// TwinCAT 3 PLC project StandardLibGema
// Title: StandardLibGema
// Company: Gema
// Author: RG
// ProjectVersion: 0.0.83
// ProgramVersion: 3.1.4024.0
// libraries:
//   RFID universal data interface TwinCAT, * (Turck)
//   Tc2_EtherCAT, * (Beckhoff Automation GmbH)
//   Tc2_Standard, * (Beckhoff Automation GmbH)
//   Tc2_System, * (Beckhoff Automation GmbH)
//   Tc2_TcpIp, * (Beckhoff Automation GmbH)
//   Tc2_Utilities, * (Beckhoff Automation GmbH)
//   Tc3_Module, * (Beckhoff Automation GmbH)
//   TcoCore, 0.11.0.71 (Vortex.Library)
//   TcoData, 0.11.0.71 (Vortex.Library)
//   TcoDrivesBeckhoff, 0.11.0.71 (Vortex.Library)
//   TcoElements, 0.11.0.71 (Vortex.Library)
//   TcoIo, 0.11.0.71 (Vortex.Library)
//   TcoPneumatics, 0.11.0.71 (Vortex.Library)
//   TcoUtilities, 0.11.0.71 (Vortex.Library)
//   TcUnit, * (www.tcunit.org)
//   BASIC,3.31,OSCAT
// project tree:
//   IAI/Data types/ AxisLimits.TcDUT, IAIAxisStatus.TcDUT, IOAxis.TcDUT (not stored)
//   IAI/Data types/Enum/ eSetPositionMode.TcDUT (not stored), E_AccelMode.TcDUT, E_RMod.TcDUT, E_StopMode.TcDUT
//   IAI/Data types/Interfaces/ iSuperActuator.TcIO (not stored)
//   IAI/Data types/In/Gateway/ GatewayStatus.TcDUT (not stored), StatusSignal0.TcDUT (not stored), StatusSignal1.TcDUT (not stored)
//   IAI/Data types/In/ PlcIn.TcDUT (not stored), StatusIn.TcDUT (not stored)
//   IAI/Data types/Out/ ControlOut.TcDUT (not stored), PlcOut.TcDUT (not stored)
//   IAI/Data types/Out/Gateway/ ControlSignal0.TcDUT (not stored), ControlSignal1.TcDUT (not stored), GatewayControl.TcDUT
//   IAI/Global Variables/ AxisStats.TcGVL (not stored), AxisStatsGlobal.TcGVL (not stored)
//   IAI/IAI_Drive/TcoAxis/ AxisIAI.TcPOU (not stored), IAxisIAI.TcIO (not stored), Power.TcPOU (not stored)
//   IAI/IAI_Drive/TcoAxis/AxisTasks/ ResetTask.TcPOU (not stored), SetPositionTask.TcPOU (not stored)
//   IAI/IAI_Drive/TcoAxis/MotionTasks/ HaltTask.TcPOU (not stored), HomeTask.TcPOU (not stored), MoveAbsoluteTask.TcPOU (not stored), MoveRelativeTask.TcPOU (not stored), StopTask.TcPOU (not stored)
//   / PlcTask.TcTTO
//   POUs/ATS400_ETL/DUT/ InputDataAts400.TcDUT, State.TcDUT
//   POUs/ATS400_ETL/FunctionBlocks/ InputAts400.TcPOU, OutputAts400.TcPOU, SelectProgramTask.TcPOU
//   POUs/ATS400_ETL/Interfaces/ IInputAts400.TcIO, IOutputAts400.TcIO
//   POUs/ATS400_ETL/Mocks/ InputAts400MockStatusReady.TcPOU
//   POUs/Communication Extern/DUTs/ E_ConnectionStepsTcp.TcDUT, OutCommunicationRobOmron.TcDUT, InCommunicationRobOmron.TcDUT, stTelegrammOmronTcp.TcDUT, uTelegrammOmronTcp.TcDUT
//   POUs/Communication Extern/FunctionBlocks/ CommunicationRoboterOmron.TcPOU, TcpIpCommSeq.TcPOU
//   POUs/Communication Extern/Interfaces/ ICommunicationRoboterOmron.TcIO, ICommSeq.TcIO
//   POUs/Counter Allgemein/ Counter.TcPOU, ICounter.TcIO, StatusCounter.TcDUT
//   POUs/Cylinders/Base/ TcoCylinderBase.TcPOU, TcoDoubleCylinderBase.TcPOU
//   POUs/Cylinders/ExampleCylinder/ ExampleCylinder.TcPOU, ExampleCylinderConfig.TcDUT, ExampleCylinderMoveTask.TcPOU, ExampleCylinderStatus.TcDUT
//   POUs/Cylinders/ ITcoCylinder.TcIO, TcoCylinder.TcPOU, TcoCylinderConfig.TcDUT, TcoCylinderMoveTask.TcPOU, TcoCylinderStatus.TcDUT, TcoDoubleCylinder.TcPOU
//   POUs/Cylinders/Zylinder/ CylCustom.TcPOU, CylCustomMoveTask.TcPOU
//   POUs/DualPositionActuator/DUTs/ E_DualPositionActuatorState.TcDUT
//   POUs/DualPositionActuator/ITFs/ I_DualPositionActuator.TcIO
//   POUs/DualPositionActuator/POUs/ FB_DualPositionActuator.TcPOU
//   POUs/Engel Ethercat Bridge Communication/DUTs/ eHeartBeatState.TcDUT, EngelInputData.TcDUT
//   POUs/Engel Ethercat Bridge Communication/FunctionBlocks/ EngelInput.TcPOU, EngelOutput.TcPOU, HeartBeat.TcPOU, IHeartBeat.TcIO, IInput.TcIO, IOutput.TcIO
//   POUs/Sequences/Test/ E_SequenceTest.TcDUT, SequenceTryout.TcPOU, stSequenceTest.TcDUT
//   POUs/SignalLights MachineStatus/DUTs/ ColorsSignalLightsStatus.TcDUT, eMachineModes.TcDUT, ColorsSignalLightMachineModes.TcDUT, eMachineStatus.TcDUT
//   POUs/SignalLights MachineStatus/ITFs/ ISignalLightsController.TcIO
//   POUs/SignalLights MachineStatus/POUs/ SignalLightsController.TcPOU
//   POUs/Turck Rfid Reader/Mock/ RfidMockNoRfidInRange.TcPOU, RfidMockWorking.TcPOU
//   POUs/Turck Rfid Reader/Rfid/ RfidHead.TcPOU, RfidInOut.TcDUT
//   POUs/Turck Rfid Reader/Rfid/Tasks/ LockTask.TcPOU, ReadDataTask.TcPOU, ReadUidTask.TcPOU, ResetTaskRfid.TcPOU, WriteDataTask.TcPOU
//   POUs/Turck Rfid Reader/Rfid/Wrapper/ IRfidHeadWrapper.TcIO, Rfid_FB_Compact_Wrapper.TcPOU
//   POUs/Utilities/ Blinker.TcPOU
//   Project Information/ F_GetCompany.TcPOU, F_GetTitle.TcPOU, F_GetVersion.TcPOU
//   Test/0 Context/ PRG_TEST.TcPOU, TcUnitContext.TcPOU, TestStation.TcPOU
//   Test/Ats400_Etl_Tests/ InputAts400_Test.TcPOU, OutputAts400_Test.TcPOU
//   Test/BlinkerTest/ Blinker_Test.TcPOU
//   Test/CommunicationExtern Tests/ CommunicationRoboterOmron_Test.TcPOU
//   Test/CounterAllgemeinTests/ Counter_Test.TcPOU
//   Test/DualPositionActuator/ FB_DualPositionActuator_Test.TcPOU
//   Test/Engel Ethercat Bridge Comm Tests/ EngelInput_Test.TcPOU, EngelOutput_Test.TcPOU, HeartBeat_Test.TcPOU
//   Test/Sequences/Test/ SequenceTryout_Test.TcPOU
//   Test/SignalLights MachineStatus Tests/ SignalLightsController_Test.TcPOU
//   Test/Turck Rfid Reader Test/ RfidHead_Test.TcPOU
//   Test/Zylinder Tests/ CylCustom_Test.TcPOU
//   Version/ Global_Version.TcGVL
// real-time tasks:
//   TASK PlcTask: cycle T#1ms, priority 20, ADS port 350

CONFIGURATION StandardLibGema
    RESOURCE PLC ON TwinCAT3
        TASK PlcTask(INTERVAL := T#1ms, PRIORITY := 20);
        PROGRAM PRG_TEST WITH PlcTask : PRG_TEST;
    END_RESOURCE
END_CONFIGURATION

// ---- IAI/Data types/AxisLimits.TcDUT
TYPE
    AxisLimits :
    STRUCT
        MaxAcceleration : UINT;
        MINPosition     : DINT;
        MaxPosition     : DINT;
        MaxVelocity     : UINT;
    END_STRUCT
END_TYPE

// ---- IAI/Data types/Enum/E_AccelMode.TcDUT
//(*Operating mode selector: The AUTO mode is selected when this
//	 signal is OFF, and the MANU mode is selected when the signal is ON*)
TYPE
    E_AccelMode :
    (
        AMode_Trapetz    := 0, (*default*)
        AMode_S_Shape    := 1,
        AMode_FirstOrder := 2
    );
END_TYPE

// ---- IAI/Data types/Enum/E_RMod.TcDUT
//(*Operating mode selector: The AUTO mode is selected when this
//	 signal is OFF, and the MANU mode is selected when the signal is ON*)
TYPE
    E_RMod :
    (
        RMode_Auto := 0,
        RMode_Manu := 1
    );
END_TYPE

// ---- IAI/Data types/Enum/E_StopMode.TcDUT
//(*Operating mode selector: The AUTO mode is selected when this
//	 signal is OFF, and the MANU mode is selected when the signal is ON*)
TYPE
    E_StopMode :
    (
        SMode_OFF      := 0,
        SMode_Param_36 := 1,
        SMode_Param_37 := 2,
        SMode_Param_38 := 3
    );
END_TYPE

// ---- IAI/Data types/IAIAxisStatus.TcDUT
{attribute wpf [Container(Layout.Wrap)]}
TYPE
    IAIAxisStatus :
    STRUCT
        {attribute wpf [Container(Layout.Stack)]}
        {attribute addProperty Name "<#Actual position in mm#>"}
        ActPos : LREAL; (* Actual position (absolut value from NC) *)
        //        {attribute addProperty Name "<#Actual modulo position#>"}
        //        ModuloActPos : LREAL; (* Actual modulo position *)
        //        {attribute addProperty Name "<#Actual modulo turns#>"}
        //        ModuloActTurns : DINT; (* Actual modulo turns *)
        {attribute addProperty Name "<#Actual velocity#>"}
        ActVelo : LREAL; (* Actual velocity *)
        {attribute addProperty Name "<#Actual acceleration#>"}
        ActAcc : LREAL;
        {attribute addProperty Name "<#Actual torque#>"}
        ActTorque : LREAL;
        //        {attribute addProperty Name "<#Command number#>"}
        //        CmdNo : WORD; (* Continuous actual command number *)
        //        {attribute addProperty Name "<#Command state#>"}
        //        CmdState : WORD; (* Command state *)
        //        {attribute addProperty Name "<#Motion state#>"}
        //        MotionState : eAxisStates; (* motion state in the PLCopen state diagram *)
        {attribute addProperty Name "<#Error#>"}
        Error : BOOL; (* axis error state *)
        {attribute addProperty Name "<#Error id#>"}
        ErrorId : UDINT; (* axis error code *)

        (* PLCopen motion control statemachine states: *)
        //        ErrorStop : BOOL;
        //        Disabled : BOOL;
        //        Stopping : BOOL;
        StandStill       : BOOL;
        DiscreteMotion   : BOOL;
        ContinuousMotion : BOOL;
        AbsoluteMotion   : BOOL;
        RelativeMotion   : bool;
        //        SynchronizedMotion : BOOL;
        Homing : BOOL;

        (* additional status - (PLCopen definition)*)
        //        ConstantVelocity : BOOL;
        //        Accelerating : BOOL;
        //        Decelerating : BOOL;

        (* Axis.NcToPlc.StateDWord *)
        Operational : BOOL;
        //        ControlLoopClosed : BOOL; (* operational and position control active *)
        //        HasJob : BOOL;
        HasBeenStopped : BOOL;
        //        NewTargetPosition : BOOL; (* new target position commanded during move *)
        {attribute wpf [Container(Layout.Stack)]}
        InPositionArea    : BOOL;
        InTargetPosition1 : BOOL;
        InTargetPosition2 : BOOL;

        Homed : BOOL;
        //        HomingBusy : BOOL;
        //        MotionCommandsLocked : BOOL; (* stop 'n hold *)
        //        SoftLimitMinExceeded : BOOL; (* reverse soft travel limit exceeded *)
        //        SoftLimitMaxExceeded : BOOL; (* forward soft travel limit exceeded *)

        Moving            : BOOL;
        PositiveDirection : BOOL;
        NegativeDirection : BOOL;
        NotMoving         : BOOL;
        //        Compensating : BOOL; (* superposition - overlayed motion *)

        //        ExtSetPointGenEnabled : BOOL;
        //        ExternalLatchValid : BOOL;
        //        CamDataQueued : BOOL;
        //        CamTableQueued : BOOL;
        //        CamScalingPending : BOOL;
        //        CmdBuffered : BOOL;
        //        PTPmode : BOOL;
        DriveDeviceError : BOOL;
        IoDataInvalid    : BOOL;

        (* Axis.NcToPlc.CoupleState *)
        Coupled1 : BOOL;
        Coupled2 : BOOL;
        Coupled3 : BOOL;
        Coupled4 : BOOL;

    //        (* axis operation mode feedback from NcToPlc *)
    //        OpMode : TcoAxisOpModes;
    END_STRUCT
END_TYPE

// ---- IAI/Data types/Out/Gateway/GatewayControl.TcDUT
TYPE
    GatewayControl :
    STRUCT
        GatewayControl0 : ControlSignal0;
        GatewayControl1 : ControlSignal1;
        RequestCmd      : WORD;
        Data0           : WORD;
        Data1           : WORD;
        Data2           : WORD;
        Data3           : WORD;
        UsedSpace       : WORD;
    END_STRUCT
END_TYPE

// ---- POUs/ATS400_ETL/DUT/InputDataAts400.TcDUT
TYPE
    InputDataAts400 :
    STRUCT
        Pass         : BOOL;
        Fail         : BOOL;
        InOp         : BOOL; // Digitale AUsgabe als Feedback einer aktiven sicherheitstechnischen Pruefung des Systems. Wechselt zwischen dne Pruefungen zwischen 1 auf 0
        ResultImpuls :
            BOOL; // Einstellbare digitale Ausgavbe eines Impuls. Z.B. Gesamtergebnis schlecht, Gesamtergebnis gut etc.
        DummyOut :
            BOOL; //Anofrderung Dummypruefung durch SPS, wartet auf weiteres Feeedback bis Dummy-Pruefobjekt bereit ist
        Ready :
            BOOL;             // wartet auf Start
        SafetyCircuit : BOOL; // 1 = closed, 0 = Open, oder externes Relais, Anzugs- oder Abfallzeit <= 200ms !!
        ContactExits  : BOOL; // Kontaktueberwachung, 1 = Kontakt vorhanden, oder externes Relais
    END_STRUCT
END_TYPE

// ---- POUs/ATS400_ETL/DUT/State.TcDUT
{attribute 'qualified_only'}
{attribute 'strict'}
TYPE
    State :
    (
        Ready := 0,
        Busy,
        Done,
        Fail
    );
END_TYPE

// ---- POUs/Communication Extern/DUTs/E_ConnectionStepsTcp.TcDUT
TYPE
    E_ConnectionStepsTcp :
    (
        eCONNECTION_STATE_IDLE,
        eCONNECTION_STATE_CONNECT_START,
        eCONNECTION_STATE_CONNECT_WAIT,
        eCONNECTION_STATE_DATAEXCHANGE,
        eCONNECTION_STATE_CLOSE_START,
        eCONNECTION_STATE_CLOSE_WAIT,
        eCONNECTION_STATE_ERROR
    );
END_TYPE

// ---- POUs/Communication Extern/DUTs/OutCommunicationRobOmron.TcDUT
TYPE
    OutCommunicationRobOmron :
    STRUCT
        {attribute addProperty Name "<#AutoMode Aktiv#>"}
        StartAutomatic  : BOOL;
        StopAutomatic   : BOOL;
        Reset           : BOOL;
        RequestHome     : BOOL;
        HighPowerOn     : BOOL;
        HighPowerOff    : BOOL;
        ContactPrepared : BOOL;
    END_STRUCT
END_TYPE

// ---- POUs/Communication Extern/DUTs/InCommunicationRobOmron.TcDUT
TYPE
    InCommunicationRobOmron :
    STRUCT
        {attribute addProperty Name "<#Home Pos erreicht#>"}
        homePosReached : BOOL;
        {attribute addProperty Name "<#Status Running#>"}
        statusRunning : BOOL;
        {attribute addProperty Name "<#Fehler#>"}
        Fault : BOOL;
        {attribute addProperty Name "<#Fehler ID#>"}
        FaultID : INT;
        {attribute addProperty Name "<#HighPower aktiv#>"}
        PowerOn : BOOL;
        {attribute addProperty Name "<#EStop aktiv#>"}
        Estop : BOOL;
    END_STRUCT
END_TYPE

// ---- POUs/Communication Extern/DUTs/stTelegrammOmronTcp.TcDUT
{attribute 'pack_mode' := '1'}
TYPE
    stTelegrammOmronTcp :
    STRUCT
        myStats  : ARRAY[1..4] OF BYTE;
        myInt    : ARRAY[1..10] OF INT;
        myBool   : ARRAY[1..20] OF INT;
        fillbyte : ARRAY[1..2] OF BYTE;
    END_STRUCT
END_TYPE

// ---- POUs/Communication Extern/DUTs/uTelegrammOmronTcp.TcDUT
TYPE
    uTelegrammOmronTcp :
    UNION
        //~
        stTel : stTelegrammOmronTcp;
        aTel  : ARRAY[1..SIZEOF(stTelegrammOmronTcp)] OF BYTE;
        sTel  : STRING(SIZEOF(stTelegrammOmronTcp));
    //~
    END_UNION
END_TYPE

// ---- POUs/Counter Allgemein/StatusCounter.TcDUT
{attribute 'qualified_only'}
{attribute 'strict'}
TYPE StatusCounter :
(
    Error := 0,
    Run,
    Unknown
);
END_TYPE

// ---- POUs/Cylinders/ExampleCylinder/ExampleCylinderConfig.TcDUT
TYPE
    ExampleCylinderConfig :
    STRUCT
        TimeToReachHomePosition : TIME := T#10S;
        TimeToReachWorkPosition : TIME := T#10S;
    END_STRUCT
END_TYPE

// ---- POUs/Cylinders/ExampleCylinder/ExampleCylinderStatus.TcDUT
TYPE
    ExampleCylinderStatus :
    STRUCT
        ActionDescription : STRING(100);
    END_STRUCT
END_TYPE

// ---- POUs/Cylinders/TcoCylinderConfig.TcDUT
TYPE
    TcoCylinderConfig :
    STRUCT
        TimeToReachHomePosition : TIME := T#10S;
        TimeToReachWorkPosition : TIME := T#10S;
        TimeToRefill            : TIME := T#1000MS;
    END_STRUCT
END_TYPE

// ---- POUs/Cylinders/TcoCylinderStatus.TcDUT
TYPE
    TcoCylinderStatus :
    STRUCT
        ActionDescription : STRING(100);
    END_STRUCT
END_TYPE

// ---- POUs/DualPositionActuator/DUTs/E_DualPositionActuatorState.TcDUT
{attribute 'qualified_only'}
{attribute 'strict'}
{attribute 'to_string'}
TYPE
    E_DualPositionActuatorState :
    (
        Unknown := 0,
        Active,
        Disabled,
        TimeoutActivating,
        TimeoutDisabling,
        Activating,
        Disabling
    ) INT;
END_TYPE

// ---- POUs/Engel Ethercat Bridge Communication/DUTs/eHeartBeatState.TcDUT
{attribute 'qualified_only'}
{attribute 'strict'}
{attribute 'to_string'}
TYPE
    eHeartBeatState :
    (
        Unknown := 0,
        Valid,
        Timeout
    ) INT;
END_TYPE

// ---- POUs/Engel Ethercat Bridge Communication/DUTs/EngelInputData.TcDUT
TYPE
    EngelInputData :
    STRUCT
        HeartBeat            : UINT;
        ManualActive         : BOOL;
        AutoActive           : BOOL;
        AutoStart            : BOOL;
        HomeRequest          : BOOL;
        HomeDone             : BOOL;
        SafetyClosed         : BOOL;
        SafetyOpeningAllowed : BOOL;

    END_STRUCT
END_TYPE

// ---- POUs/Sequences/Test/E_SequenceTest.TcDUT
{attribute 'qualified_only'}
{attribute 'strict'}
{attribute 'to_string'}
TYPE
    E_SequenceTest :
    (
        WaitForStart,
        OpenValveAandB,
        ConfirmValvesAandBOpend,
        CloseValveA,
        ConfirmClosedValveA,
        Error,
        Done
    ) INT;
END_TYPE

// ---- POUs/Sequences/Test/stSequenceTest.TcDUT
TYPE
    stSequenceTest :
    STRUCT
        WaitForStart   : INT := 10;
        OpenValveAandB : INT := 20;
    END_STRUCT
END_TYPE

// ---- POUs/SignalLights MachineStatus/DUTs/ColorsSignalLightsStatus.TcDUT
TYPE
    ColorsSignalLightsStatus :
    STRUCT
        Blue     : BOOL;
        White    : BOOL;
        Violet   : BOOL;
        Turquise : BOOL;
    END_STRUCT
END_TYPE

// ---- POUs/SignalLights MachineStatus/DUTs/eMachineModes.TcDUT
{attribute 'qualified_only'}
{attribute 'strict'}
{attribute 'to_string'}
TYPE
    eMachineModes :
    (
        Idle    := 0,
        Automat := 1000,
        Step    := 2000,
        Home    := 3000,
        Manual  := 4000,
        Fault   := 9000
    ) INT;
END_TYPE

// ---- POUs/SignalLights MachineStatus/DUTs/ColorsSignalLightMachineModes.TcDUT
TYPE
    ColorsSignalLightMachineModes :
    STRUCT
        Green       : BOOL;
        Yellow      : BOOL;
        Red         : BOOL;
    END_STRUCT
END_TYPE

// ---- POUs/SignalLights MachineStatus/DUTs/eMachineStatus.TcDUT
{attribute 'qualified_only'}
{attribute 'strict'}
{attribute 'to_string'}
TYPE
    eMachineStatus :
    (

        Blue     := 100,
        White    := 200,
        Violet   := 300,
        Turquise := 400,
        All      := 990
    ) INT;
END_TYPE

// ---- POUs/Turck Rfid Reader/Rfid/RfidInOut.TcDUT
TYPE
    RfidInOut :
    STRUCT

        myReadData             : ARRAY[0..127] OF BYTE;
        myWriteData            : ARRAY[0..127] OF BYTE;
        xExecute               : BOOL;
        xAbort                 : BOOL;
        udiTimeOut             : UDINT;
        eCommand               : RFID_FB_U.COMMAND;
        udiStartAdress         : UDINT;
        uiDataLenght           : UINT;
        xDone                  : BOOL;
        xBusy                  : BOOL;
        xError                 : BOOL;
        xAborted               : BOOL;
        eErrorID               : RFID_FB_U.ERROR;
        xTP                    : BOOL;
        xRWHeadNotCOnnected    : BOOL;
        uiDataRxLength         : UINT;
        stCompactModeInputMap  : RFID_FB_U.CompactInput_t;
        stCompactModeOutputMap : RFID_FB_U.CompactOutput_t;
    END_STRUCT
END_TYPE

// ---- Version/Global_Version.TcGVL
{attribute 'TcGenerated'}
{attribute 'no-analysis'}
{attribute 'linkalways'}
// This function has been automatically generated from the project information.
VAR_GLOBAL CONSTANT
    {attribute 'const_non_replaced'}
    stLibVersion_StandardLibGema : ST_LibVersion :=
    (
        iMajor      := 0
        , iMinor    := 0
        , iBuild    := 83
        , iRevision := 0
        , nFlags    := 0
        , sVersion  := '0.0.83'
    );
END_VAR

// ---- POUs/ATS400_ETL/Interfaces/IInputAts400.TcIO
INTERFACE IInputAts400 EXTENDS __SYSTEM.IQueryInterface

METHOD GetInputData : InputDataAts400
VAR_INPUT
END_VAR
END_METHOD

END_INTERFACE

// ---- POUs/ATS400_ETL/Interfaces/IOutputAts400.TcIO
INTERFACE IOutputAts400 EXTENDS __SYSTEM.IQueryInterface

METHOD AbortTest
VAR_INPUT
    enable : BOOL;
END_VAR
END_METHOD

METHOD SelectProgramm : TcoCore.ITcoTaskStatus
VAR_INPUT
    programm : UINT;
END_VAR
END_METHOD

METHOD SetDummyReady
VAR_INPUT
    enable : BOOL;
END_VAR
END_METHOD

METHOD SetManualFail
VAR_INPUT
    enable : BOOL;
END_VAR
END_METHOD

METHOD SetManualPass
VAR_INPUT
    enable : BOOL;
END_VAR
END_METHOD

METHOD Start
VAR_INPUT
    enable : BOOL;
END_VAR
END_METHOD

END_INTERFACE

// ---- POUs/Communication Extern/Interfaces/ICommunicationRoboterOmron.TcIO
INTERFACE ICommunicationRoboterOmron EXTENDS __SYSTEM.IQueryInterface

METHOD ContactPrepared
VAR_INPUT
    enable : BOOL;
END_VAR
END_METHOD

PROPERTY EState : E_SocketConnectionState
GET
END_GET
END_PROPERTY

METHOD HighPowerOn
VAR_INPUT
    enable : BOOL;
END_VAR
END_METHOD

PROPERTY MsgFmtStr : T_MaxString
GET
END_GET
END_PROPERTY

METHOD RequestHome
VAR_INPUT
    enable : BOOL;
END_VAR
END_METHOD

METHOD Reset
VAR_INPUT
    enable : BOOL;
END_VAR
END_METHOD

METHOD Run
END_METHOD

METHOD StartAutomatic
VAR_INPUT
    enable : BOOL;
END_VAR
END_METHOD

METHOD StopAutomatic
VAR_INPUT
    enable : BOOL;
END_VAR
END_METHOD

END_INTERFACE

// ---- POUs/Communication Extern/Interfaces/ICommSeq.TcIO
INTERFACE ICommSeq

PROPERTY EState : E_SocketConnectionState
GET
END_GET
END_PROPERTY

PROPERTY MsgFmtStr : T_MaxString
GET
END_GET
END_PROPERTY

METHOD Run
VAR_INPUT
    msgSend : REFERENCE TO uTelegrammOmronTcp;
    msgRcv  : REFERENCE TO uTelegrammOmronTcp;
END_VAR
END_METHOD

END_INTERFACE

// ---- POUs/Counter Allgemein/ICounter.TcIO
INTERFACE ICounter

METHOD CountDown
END_METHOD

PROPERTY CountLimitReached : BOOL
GET
END_GET
END_PROPERTY

METHOD CountUp
VAR_INPUT
END_VAR
END_METHOD

PROPERTY CountValue : UDINT
GET
END_GET
END_PROPERTY

PROPERTY CountZeroReached : BOOL
GET
END_GET
END_PROPERTY

METHOD ResetCount
VAR_INPUT
END_VAR
END_METHOD

END_INTERFACE

// ---- POUs/Cylinders/ITcoCylinder.TcIO
INTERFACE ITcoCylinder EXTENDS __System.IQueryInterface

PROPERTY AtHome : bool
GET
END_GET
END_PROPERTY

PROPERTY AtWork : bool
GET
END_GET
END_PROPERTY

METHOD MoveToHome : TcoCore.ITcoTaskStatus
END_METHOD

METHOD MoveToWork : TcoCore.ITcoTaskStatus
END_METHOD

(*~
	<docu>
		<summary>
			Stops cyclinder movement.
		 	<remarks>
				<note type="important">
					This method switched off the signals for the movement of the piston in both direction.
					However depending on the pnemumatics configuration the movement may contintue if designed in that way.
					THIS IS NOT A SAFETY FUCTION!
				</note>
			</remarks>
		</summary>
	</docu>
~*)
METHOD Stop : TcoCore.ITcoTaskStatus
END_METHOD

END_INTERFACE

// ---- POUs/DualPositionActuator/ITFs/I_DualPositionActuator.TcIO
INTERFACE I_DualPositionActuator

METHOD PUBLIC Activate
END_METHOD

METHOD PUBLIC Disable
END_METHOD

METHOD GetDisableTimeoutTime : TIME
END_METHOD

METHOD GetEnableTimeoutTime : TIME
END_METHOD

METHOD GetState : E_DualPositionActuatorState
END_METHOD

METHOD SetDisableTimeoutTime
VAR_INPUT
    tDisableTimeoutTime : TIME;
END_VAR
END_METHOD

METHOD SetEnableTimeoutTime
VAR_INPUT
    tEnableTimeoutTime : TIME;
END_VAR
END_METHOD

END_INTERFACE

// ---- POUs/Engel Ethercat Bridge Communication/FunctionBlocks/IHeartBeat.TcIO
INTERFACE IHeartBeat EXTENDS __SYSTEM.IQueryInterface

PROPERTY GetErrorMessage : T_MaxString;
GET
END_GET
END_PROPERTY

//actual Heartbeat of PLC
PROPERTY GetHeartBeat : UINT
GET
END_GET
END_PROPERTY

PROPERTY GetHeartbeatTimeoutTime : TIME
GET
END_GET
END_PROPERTY

PROPERTY GetState : eHeartBeatState
GET
END_GET
END_PROPERTY

METHOD IncreaseHeartBeat : UINT
VAR_INPUT
    externalHeartBeat : UINT;
END_VAR
END_METHOD

END_INTERFACE

// ---- POUs/Engel Ethercat Bridge Communication/FunctionBlocks/IInput.TcIO
INTERFACE IInput

METHOD GetInputData : EngelInputData
END_METHOD

END_INTERFACE

// ---- POUs/Engel Ethercat Bridge Communication/FunctionBlocks/IOutput.TcIO
INTERFACE IOutput EXTENDS __SYSTEM.IQueryInterface

END_INTERFACE

// ---- POUs/SignalLights MachineStatus/ITFs/ISignalLightsController.TcIO
INTERFACE ISignalLightsController

PROPERTY GetColorsSignalLightMachineModes : ColorsSignalLightMachineModes
GET
END_GET
END_PROPERTY

PROPERTY GetColorsSignalLightMachineStatus : ColorsSignalLightsStatus
GET
END_GET
END_PROPERTY

METHOD SetBlinkTime
VAR_INPUT
    blinkOnTime  : TIME;
    blinkOffTime : TIME;
END_VAR
END_METHOD

METHOD SetMachineMode : ColorsSignalLightMachineModes
VAR_INPUT
    currentMachineMode : eMachineModes ;
END_VAR
END_METHOD

METHOD SetMachineStatusOff : ColorsSignalLightsStatus
VAR_INPUT
    currentMachineStatus : eMachineStatus ;
END_VAR
END_METHOD

METHOD SetMachineStatusOn : ColorsSignalLightsStatus
VAR_INPUT
    currentMachineStatus : eMachineStatus ;
END_VAR
END_METHOD

END_INTERFACE

// ---- POUs/Turck Rfid Reader/Rfid/Wrapper/IRfidHeadWrapper.TcIO
INTERFACE IRfidHeadWrapper

METHOD Execute
VAR_INPUT
    xExecute       : BOOL;
    xAbort         : BOOL;
    udiTimeOut     : UDINT;
    eCommand       : RFID_FB_U.COMMAND;
    udiStartAdress : UDINT;
    uiDataLenght   : UINT;
    myWriteData    : ARRAY[0..127] OF BYTE;
END_VAR
VAR_OUTPUT
    myReadData          : ARRAY[0..127] OF BYTE;
    xDone               : BOOL;
    xBusy               : BOOL;
    xError              : BOOL;
    xAborted            : BOOL;
    eErrorID            : RFID_FB_U.ERROR;
    xTP                 : BOOL;
    xRWHeadNotCOnnected : BOOL;
    uiDataRxLength      : UINT;
END_VAR
END_METHOD

END_INTERFACE

// ---- Test/0 Context/PRG_TEST.TcPOU
PROGRAM PRG_TEST
VAR
    _testSuite : TcUnitContext;
END_VAR

_testSuite.Run();
_testSuite.RtcSynchronize(true, '', 60);

END_PROGRAM

// ---- Test/0 Context/TcUnitContext.TcPOU
FUNCTION_BLOCK TcUnitContext EXTENDS TcoCore.TcoContext
VAR
    testStation : TestStation(THIS^);

    {attribute addProperty Name "Versionsnummer Plc"}
    version : STRING(23);
    //~
    programVersion : ST_LibVersion;
    //~

END_VAR

(*~
    <docu>
        <summary>
            Main method of the TcoContext. This is the entry point of any control logic that belongs to this context.
            The call of this method is ensured by calling the <c>InstanceName.Run()</c> method, and it must not be called explicitly.
            This method is abstract, and it must be overridden in derived block.
        </summary>
    </docu>
~*)
METHOD PROTECTED Main

testStation();
END_METHOD

END_FUNCTION_BLOCK

// ---- Test/0 Context/TestStation.TcPOU
FUNCTION_BLOCK TestStation EXTENDS TcoCore.TcoObject
VAR
    cylCustomTest : CylCustom_Test;
END_VAR
//===============================Turck Rfid Reader===============================================
VAR
    rfidHead_Test : RfidHead_Test;
END_VAR
//===================================================================================

//====================== Engel Communication Ethercat Bridge =====================================
VAR
    engelInputTest     : EngelInput_Test;
    engelOutputTest    : EngelOutput_Test;
    engelHeartBeatTest : HeartBeat_Test;
END_VAR
//===================================================================================

//===============================Dual Position Actuator Sagatowski===============================================
VAR
    sequenceTryOutTest : SequenceTryout_Test;
END_VAR
//====
//===============================Dual Position Actuator Sagatowski===============================================
VAR
    dualPositionActuator_Test : FB_DualPositionActuator_Test;
END_VAR
//===================================================================================

//===============================Communication with ETL ATS400 ===============================================
VAR
    inputAts400Test  : InputAts400_Test;
    outputAts400Test : OutputAts400_Test;
END_VAR
//===================================================================================
//===============================Communication with ETL ATS400 ===============================================
VAR
    CommunicationRoboterOmron  : CommunicationRoboterOmron_Test;

END_VAR
//===================================================================================
//===============================SignalLights for MachineStatus ===============================================
VAR
    signalLightsControllerTest : SignalLightsController_Test;
END_VAR
//===================================================================================
//===============================Utilities ===============================================
VAR
    blinkerTest : Blinker_Test;
    counterTest : Counter_Test;
END_VAR
//=======

TcUnit.RUN();

END_FUNCTION_BLOCK

// ---- Test/Zylinder Tests/CylCustom_Test.TcPOU
FUNCTION_BLOCK CylCustom_Test EXTENDS TcUnit.FB_TestSuite IMPLEMENTS TcoCore.ITcoContext
VAR
    //Context for TcOpen
    _nfContext : TcoCore.TcoContextNfCompatibility;
END_VAR

VAR
    fbTestTimer : TON := (PT := T#30ms);
    cyl         : TcoCylinder(THIS^);
    sensor      : ARRAY[0..1] OF BOOL;
    actuator    : ARRAY[0..1] OF BOOL;
    nTestState  : INT;
END_VAR

_nfContext.VolatileOpen(); //Required for TCopen
//==============================================

ExecuteMoveToWork_SignalAtWorkShouldBeTrue();

//==============================================
_nfContext.VolatileClose();

PROPERTY Context : TcoCore.ITcoContext
GET
Context := This^._nfContext;
END_GET
END_PROPERTY

PROPERTY EndCycleCount : ULINT
GET
EndCycleCount := THIS^._nfContext._endCycleCount;
END_GET
END_PROPERTY

PROPERTY Environment : TcoCore.ITcoContextEnvironment
GET
Environment := THIS^._nfContext._settings;
END_GET
END_PROPERTY

METHOD PRIVATE ExecuteMoveToWork_SignalAtWorkShouldBeTrue
Test('ExecuteMoveToWork_SignalAtWorkShouldBeTrue');
fbTestTimer(IN := TRUE);
cyl
(
    inoAtHomePos   := sensor[0]
    , inoAtWorkPos := sensor[1]
    , inoToHomePos := actuator[0]
    , inoToWorkPos := actuator[1]
);

CASE nTestState OF
    0:
        sensor[0]  := TRUE;
        nTestState := nTestState + 1;
    1:
        // Retracted
        AssertTrue(cyl.AtHome, 'Should be AtHome');
        nTestState := nTestState + 1;
    2:
        sensor[0] := FALSE;
        cyl.MoveToWork();
        nTestState := nTestState + 1;
    3:
        AssertTrue(actuator[1], 'should turn True');
        nTestState := nTestState + 1;
    4:
        sensor[1]  := TRUE;
        nTestState := nTestState + 1;
    5:
        AssertTrue(cyl.AtWork, 'should reach Work');
END_CASE

IF fbTestTimer.Q THEN
    Assertequals_INT(Expected := 5, Actual := nTestState, Message := 'Didnt reach the last state');
    TEST_FINISHED();
END_IF
END_METHOD

PROPERTY Identity : ULINT
GET
Identity := THIS^._nfContext._Identity;
END_GET
END_PROPERTY

PROPERTY Logger : TcoCore.ITcoLogger
GET
Logger := THIS^._nfContext._logger;
END_GET
END_PROPERTY

PROPERTY RealTimeClock : TcoCore.ITcoRtc
GET
RealTimeClock := THIS^._nfContext._rtc;
END_GET
END_PROPERTY

PROPERTY StartCycleCount : ULINT
GET
StartCycleCount := THIS^._nfContext._startCycleCount;
END_GET
END_PROPERTY

END_FUNCTION_BLOCK

// ---- POUs/Cylinders/TcoCylinder.TcPOU
{attribute addProperty _moveHomeDefaultName "<#MOVE HOME#>"}
{attribute addProperty _moveWorkDefaultName "<#MOVE TO WORK#>"}
{attribute addProperty _stopDefaultName "<#STOP#>"}
FUNCTION_BLOCK TcoCylinder EXTENDS TcoCylinderBase
VAR
    {attribute addProperty Name "|[[1]Attribute_moveHomeDefaultName]|"}
    _moveHomeDefault : TcoCylinderMoveTask(THIS^);
    {attribute addProperty Name "|[[1]Attribute_moveWorkDefaultName]|"}
    _moveWorkDefault : TcoCylinderMoveTask(THIS^);
    {attribute addProperty Name "|[[1]Attribute_stopDefaultName]|"}
    _stopDefault : TcoCore.TcoTask(THIS^);
    increment    : INT;
END_VAR
VAR
    _config      : TcoCylinderConfig;
    _status      : TcoCylinderStatus;
    _refillTimer : TON;
END_VAR

SUPER^
(
    inoAtHomePos   := inoAtHomePos
    , inoAtWorkPos := inoAtWorkPos
    , inoToHomePos := inoToHomePos
    , inoToWorkPos := inoToWorkPos
);

IF (_atHomePos AND _atWorkPos) THEN
    Messenger.Error('<#Home and work position sensors are both active. Check the position of sensors!#>');
END_IF;

// Disables mutualy exclusive actions
_moveWorkDefault.Enabled := TRUE; // NOT _moveHomeDefault.Busy;

_moveHomeDefault
(
    PositionSensor           := _atHomePos AND NOT _atWorkPos
    , MoveToPositionSignal   := _toHomePos
    , InverseSignal          := _toWorkPos
    , TimeToRefill           := _config.TimeToRefill
    , MaxTimeToReachPosition := _config.TimeToReachHomePosition
    , PositionName           := '<#Home#>'
);

IF _moveHomeDefault.Execute() THEN
    _moveWorkDefault.Restore();
END_IF

// Disables mutualy exclusive actions
_moveHomeDefault.Enabled := TRUE; //NOT _moveWorkDefault.Busy;

_moveWorkDefault
(
    PositionSensor           := _atWorkPos AND NOT _atHomePos
    , MoveToPositionSignal   := _toWorkPos
    , InverseSignal          := _toHomePos
    , TimeToRefill           := _config.TimeToRefill
    , MaxTimeToReachPosition := _config.TimeToReachWorkPosition
    , PositionName           := '<#Work#>'
);

IF _moveWorkDefault.Execute() THEN
    _moveHomeDefault.Restore();
END_IF

IF (_stopDefault.Execute()) THEN
    _toHomePos := FALSE;
    _toWorkPos := FALSE;
    _moveHomeDefault.Abort();
    _moveWorkDefault.Abort();
    _stopDefault.Abort();
    _moveHomeDefault.Restore();
    _moveWorkDefault.Restore();
    _stopDefault.Restore();
    _stopDefault.DoneWhen(TRUE);
END_IF

// For further discussion about Status
IF (_moveHomeDefault.Busy) THEN
    _status.ActionDescription := 'Moving to home position';
ELSIF (_moveWorkDefault.Busy) THEN
    _status.ActionDescription := 'Moving to work position';
ELSIF (_stopDefault.Busy) THEN
    _status.ActionDescription := 'Stopping pressure';
ELSE
    _status.ActionDescription := 'Idle';
END_IF

SUPER^
(
    inoAtHomePos   := inoAtHomePos
    , inoAtWorkPos := inoAtWorkPos
    , inoToHomePos := inoToHomePos
    , inoToWorkPos := inoToWorkPos
);

(*~
    <docu>
        <summary>
            Aborts the movement to home position when the condition is 'true'.
        </summary>
        <remarks>
                <note type="warning">
                    The call of this method will be effective only when called AFTER the initialization of the instance of given TcoCylinder.
                </note>
        </remarks>
    </docu>
~*)
METHOD AbortMoveHome : BOOL
VAR_IN_OUT
    (*~
    <docu>
        <summary>
            Condition to abort the movement of the cylinder.
        </summary>
    </docu>
    ~*)
    inoDisableCondition : BOOL;
END_VAR
VAR
    _signalInfo : TcoSignalInfo;
END_VAR
IF (_toHomePos OR _moveHomeDefault.Busy) AND inoDisableCondition THEN
    _signalInfo.GetSignalInfo(SIZEOF(inoDisableCondition), ADR(inoDisableCondition));
    Messenger.Build().Append('<#Movement aborted due to#> : ').Append(_signalInfo.SymbolPath).As().AsError().Pin();
    _toHomePos := FALSE;
    IF (__ISVALIDREF(THIS^.inoToHomePos)) THEN
        THIS^.inoToHomePos := FALSE;
    END_IF;

    _moveHomeDefault.Abort();
END_IF
END_METHOD

(*~
    <docu>
        <summary>
            Aborts the movement to work position when the condition is 'true'.
        </summary>
        <remarks>
                <note type="warning">
                    The call of this method will be effective only when called AFTER the initialization of the instance of given TcoCylinder.
                </note>
        </remarks>
    </docu>
~*)
METHOD AbortMoveWork : BOOL
VAR_IN_OUT
    (*~
        <docu>
            <summary>
                Condition to abort the movement of the cylinder.
            </summary>
        </docu>
    ~*)
    inoDisableCondition : BOOL;
END_VAR
VAR
    _signalInfo : TcoSignalInfo;
END_VAR
IF (_toWorkPos OR _moveWorkDefault.Busy) AND inoDisableCondition THEN
    _signalInfo.GetSignalInfo(SIZEOF(inoDisableCondition), ADR(inoDisableCondition));
    Messenger.Build().Append('<#Movement aborted due to#> : ').Append(_signalInfo.SymbolPath).As().AsError().Pin();
    _toWorkPos := FALSE;
    IF (__ISVALIDREF(THIS^.inoToWorkPos)) THEN
        THIS^.inoToWorkPos := FALSE;
    END_IF;

    _moveWorkDefault.Abort();
END_IF
END_METHOD

(*~
    <docu>
        <summary>
            Gets the configuration of the cylinder.
        </summary>
    </docu>
~*)
PROPERTY Config : REFERENCE TO TcoCylinderConfig
GET
Config REF= _config;
END_GET
END_PROPERTY

(*~
    <docu>
        <summary>
            Gets the `MoveHomeTask` task that controls the moving of the cyclinder in home position.
        </summary>
    </docu>
~*)
PROPERTY MoveHomeTask : TcoCore.ITcoTask
GET
MoveHomeTask := _moveHomeDefault;
END_GET
END_PROPERTY

(*~
    <docu>
        <summary>
            Gets the `MoveWorkTask` task that controls the moving of the cyclinder into work position.
        </summary>
    </docu>
~*)
PROPERTY MoveWorkTask : TcoCore.ITcoTask
GET
MoveWorkTask := _moveWorkDefault;
END_GET
END_PROPERTY

(*~
    <docu>
        <summary>
            Refill cylinder after booth outputs are off .
        </summary>
        <remarks>
                <note type="warning">
                    The call of this method will be effective only when called AFTER the initialization of the instance of given TcoCylinder and methods like AbortMoveHone,SuspendMoveHom...
                </note>
        </remarks>
    </docu>
~*)
METHOD Refill : BOOL
VAR_INPUT
    (*~
    <docu>
        <summary>
            Time of refill cylinder after aborting or suspending
        </summary>
    </docu>
    ~*)
    inRefillTime : TIME;
END_VAR

_refillTimer(In := inoToHomePos XOR inoToWorkPos, Pt := T#49D);

_config.TimeToRefill := inRefillTime;

IF _refillTimer.ET > T#0MS
       AND _refillTimer.ET < _config.TimeToRefill
       AND _config.TimeToRefill <> T#0S THEN
    _toHomePos := TRUE;
    _toWorkPos := TRUE;
END_IF;

SUPER^
(
    inoAtHomePos   := inoAtHomePos
    , inoAtWorkPos := inoAtWorkPos
    , inoToHomePos := inoToHomePos
    , inoToWorkPos := inoToWorkPos
);
END_METHOD

PROPERTY StatusCom : REFERENCE TO TcoCylinderStatus
GET
StatusCom REF= _status;
END_GET
END_PROPERTY

(*~
    <docu>
        <summary>
            Gets the `StopTask` task that controls the stopping of the cyclinder.
        </summary>
    </docu>
~*)
PROPERTY StopTask : TcoCore.ITcoTask
GET
StopTask := _stopDefault;
END_GET
END_PROPERTY

(*~
    <docu>
        <summary>
            Suspend the movement to home position when the condition is 'true'. Task is still busy
        </summary>
        <remarks>
                <note type="warning">
                    The call of this method will be effective only when called AFTER the initialization of the instance of given TcoCylinder.
                </note>
        </remarks>
    </docu>
~*)
METHOD SuspendMoveHome : BOOL
VAR_IN_OUT
    (*~
    <docu>
        <summary>
            Condition to abort the movement of the cylinder.
        </summary>
    </docu>
    ~*)
    inoDisableCondition : BOOL;
END_VAR
VAR
    _signalInfo : TcoSignalInfo;
END_VAR
IF (_toHomePos OR _moveHomeDefault.Busy) AND inoDisableCondition THEN
    _signalInfo.GetSignalInfo(SIZEOF(inoDisableCondition), ADR(inoDisableCondition));
    Messenger.Warning(CONCAT('<#Movement suspended due to#> : ', _signalInfo.SymbolPath));
    _toHomePos := FALSE;
    IF (__ISVALIDREF(THIS^.inoToHomePos)) THEN
        THIS^.inoToHomePos := FALSE;
    END_IF;

END_IF
END_METHOD

METHOD SuspendMoveHomeExpression : BOOL
VAR_INPUT
    inDisableCondition : BOOL;
    inMessage          : STRING;
END_VAR
IF (_toHomePos OR _moveHomeDefault.Busy) AND inDisableCondition THEN
    Messenger.Warning(CONCAT('<#Movement suspended due to#> : ', inMessage));
    _toHomePos := FALSE;
    IF (__ISVALIDREF(THIS^.inoToHomePos)) THEN
        THIS^.inoToHomePos := FALSE;
    END_IF;

END_IF;
END_METHOD

(*~
    <docu>
        <summary>
            Suspend the movement to home position when the condition is NOT 'true'. Task is still busy
        </summary>
        <remarks>
                <note type="warning">
                    The call of this method will be effective only when called AFTER the initialization of the instance of given TcoCylinder.
                </note>
        </remarks>
    </docu>
~*)
METHOD SuspendMoveHomeInverted : BOOL
VAR_IN_OUT
    (*~
    <docu>
        <summary>
            Condition to abort the movement of the cylinder.
        </summary>
    </docu>
    ~*)
    inoDisableCondition : BOOL;
END_VAR
VAR
    _signalInfo : TcoSignalInfo;
END_VAR
IF (_toHomePos OR _moveHomeDefault.Busy) AND not inoDisableCondition THEN
    _signalInfo.GetSignalInfo(SIZEOF(inoDisableCondition), ADR(inoDisableCondition));
    Messenger.Warning(CONCAT('<#Movement suspended due to NOT#> : ', _signalInfo.SymbolPath));
    _toHomePos := FALSE;
    IF (__ISVALIDREF(THIS^.inoToHomePos)) THEN
        THIS^.inoToHomePos := FALSE;
    END_IF;

END_IF
END_METHOD

(*~
    <docu>
        <summary>
            Suspend the movement to work position when the condition is 'true'. Task is still bussy
        </summary>
        <remarks>
                <note type="warning">
                    The call of this method will be effective only when called AFTER the initialization of the instance of given TcoCylinder.
                </note>
        </remarks>
    </docu>
~*)
METHOD SuspendMoveWork : BOOL
VAR_IN_OUT
    (*~
        <docu>
            <summary>
                Condition to abort the movement of the cylinder.
            </summary>
        </docu>
    ~*)
    inoDisableCondition : BOOL;
END_VAR
VAR
    _signalInfo : TcoSignalInfo;
END_VAR
IF (_toWorkPos OR _moveWorkDefault.Busy) AND inoDisableCondition THEN
    _signalInfo.GetSignalInfo(SIZEOF(inoDisableCondition), ADR(inoDisableCondition));
    Messenger.Warning(CONCAT('<#Movement suspended due to#> : ', _signalInfo.SymbolPath));
    _toWorkPos := FALSE;
    IF (__ISVALIDREF(THIS^.inoToWorkPos)) THEN
        THIS^.inoToWorkPos := FALSE;
    END_IF;

END_IF
END_METHOD

METHOD SuspendMoveWorkExpression : BOOL
VAR_INPUT
    inDisableCondition : BOOL;
    inMessage          : STRING;
END_VAR
IF (_toWorkPos OR _moveWorkDefault.Busy) AND inDisableCondition THEN
    Messenger.Warning(CONCAT('<#Movement suspended due to#> : ', inMessage));
    _toWorkPos := FALSE;
    IF (__ISVALIDREF(THIS^.inoToWorkPos)) THEN
        THIS^.inoToWorkPos := FALSE;
    END_IF;

END_IF
END_METHOD

(*~
    <docu>
        <summary>
            Suspend the movement to work position when the condition is NOT 'true'. Task is still busy
        </summary>
        <remarks>
                <note type="warning">
                    The call of this method will be effective only when called AFTER the initialization of the instance of given TcoCylinder.
                </note>
        </remarks>
    </docu>
~*)
METHOD SuspendMoveWorkInverted : BOOL
VAR_IN_OUT
    (*~
        <docu>
            <summary>
                Condition to abort the movement of the cylinder.
            </summary>
        </docu>
    ~*)
    inoDisableCondition : BOOL;
END_VAR
VAR
    _signalInfo : TcoSignalInfo;
END_VAR
IF (_toWorkPos OR _moveWorkDefault.Busy) AND not inoDisableCondition THEN
    _signalInfo.GetSignalInfo(SIZEOF(inoDisableCondition), ADR(inoDisableCondition));
    Messenger.Warning(CONCAT('<#Movement suspended due to NOT#> : ', _signalInfo.SymbolPath));
    _toWorkPos := FALSE;
    IF (__ISVALIDREF(THIS^.inoToWorkPos)) THEN
        THIS^.inoToWorkPos := FALSE;
    END_IF;

END_IF
END_METHOD

END_FUNCTION_BLOCK

// ---- POUs/Cylinders/Base/TcoCylinderBase.TcPOU
FUNCTION_BLOCK ABSTRACT TcoCylinderBase EXTENDS TcoCore.TcoComponent IMPLEMENTS ITcoCylinder
VAR_IN_OUT
    (*~
        <docu>
            <summary>
                Home position sensor.
            </summary>
        </docu>
    ~*)
    {attribute addProperty Name "<#Home position sensor#>"}
    inoAtHomePos : BOOL;
    (*~
        <docu>
            <summary>
                Working position sensor.
            </summary>
        </docu>
    ~*)
    {attribute addProperty Name "<#Work position sensor#>"}
    inoAtWorkPos : BOOL;
END_VAR
VAR_IN_OUT
    (*~
        <docu>
            <summary>
                Move to working home position signal.
            </summary>
        </docu>
    ~*)
    {attribute addProperty Name "<#Move to home position actuator#>"}
    inoToHomePos : BOOL;
    (*~
        <docu>
            <summary>
                Move to working posistion signal.
            </summary>
        </docu>
    ~*)
    {attribute addProperty Name "<#Move to work position actuator#>"}
    inoToWorkPos : BOOL;
END_VAR
VAR
    (*~
        <docu>
            <summary>
                Home position sensor.
            </summary>
        </docu>
    ~*)
    {attribute addProperty Name "<#Home position sensor#>"}
    _atHomePos : BOOL;
    (*~
        <docu>
            <summary>
                Working position sensor.
            </summary>
        </docu>
    ~*)
    {attribute addProperty Name "<#Work position sensor#>"}
    _atWorkPos : BOOL;
    (*~
        <docu>
            <summary>
                Move to working home position signal.
            </summary>
        </docu>
    ~*)
    {attribute addProperty Name "<#Move to home position actuator#>"}
    _toHomePos : BOOL;
    (*~
        <docu>
            <summary>
                Move to working posistion signal.
            </summary>
        </docu>
    ~*)
    {attribute addProperty Name "<#Move to work position actuator#>"}
    _toWorkPos : BOOL;
END_VAR

VAR
    {attribute addProperty Name "<#Home sensor signal#>"}
    _atHomePosSignalInfo : TcoCore.TcoSignalInfo;
    {attribute addProperty Name "<#Work sensor signal#>"}
    _atWorkPosSignalInfo : TcoCore.TcoSignalInfo;
    {attribute addProperty Name "<#Move to home position signal#>"}
    _toHomePosSignalInfo : TcoCore.TcoSignalInfo;
    {attribute addProperty Name "<#Move to work position signal#>"}
    _toWorkPosSignalInfo : TcoCore.TcoSignalInfo;
END_VAR

IF (__ISVALIDREF(inoAtHomePos)) THEN
    _atHomePos := inoAtHomePos;
    _atHomePosSignalInfo.GetSignalInfo(SIZEOF(inoAtHomePos), ADR(inoAtHomePos));
END_IF;

IF (__ISVALIDREF(inoAtWorkPos)) THEN
    _atWorkPos := inoAtWorkPos;
    _atWorkPosSignalInfo.GetSignalInfo(SIZEOF(inoAtWorkPos), ADR(inoAtWorkPos));
END_IF;

IF (__ISVALIDREF(inoToHomePos)) THEN
    inoToHomePos := _toHomePos;
    _toHomePosSignalInfo.GetSignalInfo(SIZEOF(inoToHomePos), ADR(inoToHomePos));
END_IF;

IF (__ISVALIDREF(inoToWorkPos)) THEN
    inoToWorkPos := _toWorkPos;
    _toWorkPosSignalInfo.GetSignalInfo(SIZEOF(inoToWorkPos), ADR(inoToWorkPos));
END_IF;

(*~
    <docu>
        <summary>
            Gets whether the piston is in home position.
        </summary>
    </docu>
~*)
PROPERTY AtHome : bool
GET
AtHome := THIS^._atHomePos;
END_GET
END_PROPERTY

(*~
    <docu>
        <summary>
            Gets whether the piston is in work position.
        </summary>
    </docu>
~*)
PROPERTY AtWork : bool
GET
AtWork := _atWorkPos;
END_GET
END_PROPERTY

METHOD FB_init : BOOL
VAR_INPUT
    bInitRetains : BOOL; // if TRUE, the retain variables are initialized (warm start / cold start)
    bInCopyCode  : BOOL; // if TRUE, the instance afterwards gets moved into the copy code (online change)
    ParentObject : ITcoObject;
END_VAR
END_METHOD

(*~
    <docu>
        <summary>
            Gets the `MoveHomeTask` task that controls the moving of the cyclinder in home position.
            <remarks>
                <note type="important">
                    This is an abstract method and must be implemented in derived class.
                </note>
            </remarks>
        </summary>
    </docu>
~*)
PROPERTY PUBLIC ABSTRACT MoveHomeTask : TcoCore.ITcoTask
GET
END_GET
END_PROPERTY

(*~
    <docu>
        <summary>
            Starts movement into home position.
        </summary>
    </docu>
~*)
METHOD MoveToHome : TcoCore.ITcoTaskStatus
IF (MoveHomeTask <> 0) THEN
    MoveToHome := MoveHomeTask.Invoke();
END_IF;
END_METHOD

(*~
    <docu>
        <summary>
            Starts movement into work position.
        </summary>
    </docu>
~*)
METHOD MoveToWork : TcoCore.ITcoTaskStatus
IF (MoveWorkTask <> 0) THEN
    MoveToWork := MoveWorkTask.Invoke();
END_IF;
END_METHOD

(*~
    <docu>
        <summary>
            Gets the `MoveWorkTask` task that controls the moving of the cyclinder into work position.
            <remarks>
                <note type="important">
                    This is an abstract method and must be implemented in derived class.
                </note>
            </remarks>
        </summary>
    </docu>
~*)
PROPERTY PUBLIC ABSTRACT MoveWorkTask : TcoCore.ITcoTask
GET
END_GET
END_PROPERTY

(*~
    <docu>
        <summary>
            Restore all tasks of this instance into initial state.
        </summary>
    </docu>
~*)
METHOD Restore : ITcoRestorable
IF (MoveHomeTask <> 0) THEN
    MoveHomeTask.Restore();
END_IF;

IF (MoveWorkTask <> 0) THEN
    MoveWorkTask.Restore();
END_IF;

IF (StopTask <> 0) THEN
    StopTask.Restore();
END_IF;
END_METHOD

METHOD PROTECTED ServiceMode
END_METHOD

(*~
    <docu>
        <summary>
            Stops cyclinder movement.
             <remarks>
                <note type="important">
                    This method switched off the signals for the movement of the piston in both direction.
                    However depending on the pnemumatics configuration the movement may contintue if designed in that way.
                    THIS IS NOT A SAFETY FUCTION!
                </note>
            </remarks>
        </summary>
    </docu>
~*)
METHOD Stop : TcoCore.ITcoTaskStatus
IF (StopTask <> 0) THEN
    Stop := StopTask.Invoke();
END_IF;
END_METHOD

(*~
    <docu>
        <summary>
            Gets the `StopTask` task that controls the stopping cyclinder movement.
            <remarks>
                <note type="important">
                    This is an abstract method and must be implemented in derived class.
                </note>
            </remarks>
        </summary>
    </docu>
~*)
PROPERTY PUBLIC ABSTRACT StopTask : TcoCore.ITcoTask
GET
END_GET
END_PROPERTY

END_FUNCTION_BLOCK

// ---- POUs/Cylinders/TcoCylinderMoveTask.TcPOU
FUNCTION_BLOCK TcoCylinderMoveTask EXTENDS TcoCore.TcoTask
VAR_INPUT
    PositionSensor         : BOOL;
    MaxTimeToReachPosition : TIME := T#10S;
    TimeToRefill           : TIME := T#100MS;
    PositionName           : STRING(25);
END_VAR
VAR_IN_OUT
    MoveToPositionSignal : BOOL;
    InverseSignal        : BOOL;
END_VAR

VAR
    _stringBuilder : TcoCore.StringBuilder;
END_VAR

IF (THIS^.Execute()) THEN
    IF (THIS^.ElapsedTime > MaxTimeToReachPosition) THEN
        THIS^.Messenger
            .Warning(_stringBuilder.Clear().Append(PositionName).Append(' sensor not reached yet.').ToString());
    END_IF;

    InverseSignal        := FALSE;
    MoveToPositionSignal := TRUE;
    THIS^.DoneWhen(PositionSensor);
END_IF

METHOD PUBLIC FB_init : BOOL
VAR_INPUT
    bInitRetains : BOOL; // if TRUE, the retain variables are initialized (warm start / cold start)
    bInCopyCode  : BOOL; // if TRUE, the instance afterwards gets moved into the copy code (online change)
    ParentObject : ITcoObject;
END_VAR
END_METHOD

(*~
    <docu>
        <summary>
            Executes when task is aborted.
        </summary>
    </docu>
~*)
METHOD PROTECTED OnAbort
MoveToPositionSignal := FALSE;
END_METHOD

METHOD PROTECTED OnError
END_METHOD

METHOD PROTECTED OnStart
END_METHOD

END_FUNCTION_BLOCK

// ---- Test/Turck Rfid Reader Test/RfidHead_Test.TcPOU
FUNCTION_BLOCK RfidHead_Test EXTENDS TcUnit.FB_TestSuite IMPLEMENTS TcoCore.ITcoContext
VAR
    //Context for TcOpen
    _nfContext : TcoCore.TcoContextNfCompatibility;
END_VAR
VAR
    _wrapper_RfidMockNoRfidInRange : RfidMockNoRfidInRange;

    sut_readDataNoTag                  : RfidHead(THIS^, _wrapper_RfidMockNoRfidInRange, T#10MS);
    sut_readUidNoTag                   : RfidHead(THIS^, _wrapper_RfidMockNoRfidInRange, T#10MS);
    _wrapper_readUid                   : RfidMockWorking;
    sut_readUidSuccess                 : RfidHead(THIS^, _wrapper_readUid, T#10MS);
    _wrapper_readData                  : RfidMockWorking;
    sut_readDataSuccess                : RfidHead(THIS^, _wrapper_readData, T#10MS);
    _wrapper_RfidMockTooLong           : RfidMockWorking;
    sut_readDataTooLongString          : RfidHead(THIS^, _wrapper_RfidMockTooLong, T#10MS);
    _wrapper_writeData                 : RfidMockWorking;
    sut_writeDataSuccess               : RfidHead(THIS^, _wrapper_writeData, T#10MS);
    _wrapper_readDataWithOffset        : RfidMockWorking;
    sut_readDataWithOffset             : RfidHead(THIS^, _wrapper_readDataWithOffset, T#10MS);
    _wrapper_writeDataWithOffset       : RfidMockWorking;
    sut_writeDataWithOffsetSuccess     : RfidHead(THIS^, _wrapper_writeDataWithOffset, T#10MS);
    _wrapper_readDataWithOffsetTooLong : RfidMockWorking;
    sut_readDataWithOffsetTooLong      : RfidHead(THIS^, _wrapper_readDataWithOffsetTooLong, T#10MS);
    _wrapper_lock                      : RfidMockWorking;
    sut_lockSuccess                    : RfidHead(THIS^, _wrapper_lock, T#10MS);
    _wrapper_RfidMockCreateError       : RfidMockWorking;
    sut_readDataCreateEmptyString      : RfidHead(THIS^, _wrapper_RfidMockCreateError, T#10MS);

END_VAR

_nfContext.VolatileOpen(); //Required for TCopen
//==============================================

//
ExecuteReadDataWithTooLongDataLength_ExpectErrorWithErroId();
ExecuteReadDataWithOffsetTooHigh_ExpectErrorWithErroId();
//
ExecuteReadUidsNoTagInRange_ExpectErrorWithNoTag();
ExecuteReadDataNoTagInRange_ExpectErrorWithNoTag();

//
ExecuteReadUid_ExpectUidAsStringStatusDone();
ExecuteReadData_ExpectDataAsStringStatusDone();
ExecuteReadDataWithOffset_ExpectDataAsString();

//
ExecuteWriteData_ExpectStatusDone();
ExecuteReadDataWrongParameter_ExpectErrorAndStringError();
// Lock testen,
// Locken, muss Status done, Schreiben mit Error
ExecuteLock_ExpectStatusDone();
//==============================================
_nfContext.VolatileClose();

PROPERTY Context : TcoCore.ITcoContext
GET
Context := This^._nfContext;
END_GET
END_PROPERTY

PROPERTY EndCycleCount : ULINT
GET
EndCycleCount := THIS^._nfContext._endCycleCount;
END_GET
END_PROPERTY

PROPERTY Environment : TcoCore.ITcoContextEnvironment
GET
Environment := THIS^._nfContext._settings;
END_GET
END_PROPERTY

METHOD PRIVATE ExecuteLock_ExpectStatusDone
VAR_INST
    _udiDataLength : UINT := 4;
    _offSet        : BYTE := 1;
    _result        : BOOL;

    _first : BOOL := TRUE;
END_VAR
TcUnit.TEST('ExecuteLock_ExpectStatusDone');
//Arrange
sut_lockSuccess();

//Act
sut_lockSuccess.LockMethod(udiDataLength := _udiDataLength, StartAdress := _offSet);

_result := TRUE;

//Needs two Cycles to get from Status Requested to Buisy (TcOpen Framework)
sut_lockSuccess();

IF _first THEN
    AssertEquals_BOOL
    (
        Expected  := _result
        , Actual  := sut_lockSuccess.pLockTask.Busy
        , Message := 'Status Busy muss true sein'
    );

    _first := FALSE;
END_IF

IF sut_lockSuccess.pLockTask.Done THEN

    _result := FALSE;
    AssertEquals_BOOL
    (
        Expected  := _result
        , Actual  := sut_lockSuccess.pLockTask.Busy
        , Message := 'Status Busy muss false sein'
    );

    _result := TRUE;
    AssertEquals_BOOL
    (
        Expected  := _result
        , Actual  := sut_lockSuccess.LockMethod(udiDataLength := _udiDataLength, StartAdress := _offSet).Done
        , Message := 'Status Done muss true sein'
    );

    TcUnit.TEST_FINISHED();
END_IF
END_METHOD

METHOD PRIVATE ExecuteReadData_ExpectDataAsStringStatusDone
VAR_INST
    _data          : T_MaxString;
    _expectedData  : T_MaxString := '16# 05 06 07 08';
    _result        : BOOL;
    _udiDataLength : uINT := 4;
END_VAR
//{warning disable C0371}
TcUnit.TEST('ExecuteReadData_ExpectDataAsStringStatusDone');
//Arrange
sut_readDataSuccess();

//Act

sut_readDataSuccess.ReadDataMethod(_udiDataLength, 0);
//Assert

IF sut_readDataSuccess.pReadDataTask.Done THEN
    _data := sut_readDataSuccess.Data;

    AssertEquals_STRING(Expected := _expectedData, Actual := _data, Message := 'Daten passt nicht');

    //Busy off
    _result := FALSE;
    AssertEquals_BOOL
    (
        Expected  := _result
        , Actual  := sut_readDataSuccess.pReadDataTask.Busy
        , Message := 'Status Busy muss false sein'
    );

    //Status Done mus True sein
    _result := true;
    AssertEquals_BOOL
    (
        Expected  := _result
        , Actual  := sut_readDataSuccess.ReadDataMethod(_udiDataLength, 0).Done
        , Message := 'Status Done muss true sein'
    );

    //Status Done false again
    sut_readDataSuccess.Restore();
    _result := FALSE;
    AssertEquals_BOOL
    (
        Expected  := _result
        , Actual  := sut_readDataSuccess.ReadDataMethod(_udiDataLength, 0).Done
        , Message := 'Status Done muss false sein nach Reset'
    );

    TcUnit.TEST_FINISHED();
END_IF
END_METHOD

METHOD PRIVATE ExecuteReadDataNoTagInRange_ExpectErrorWithNoTag
VAR_INST
    _udiDataLength : uINT := 3;
    _result        : BOOL;
    _firstRun      : BOOL := TRUE;

    _expectedErrorId : RFID_FB_U.ERROR;
    _errorId         : RFID_FB_U.ERROR;

END_VAR
TcUnit.TEST('ExecuteReadDataNoTagInRange_ExpectErrorWithNoTag');

//Assert Initial State
_result := FALSE;

IF _firstRun THEN
    _firstRun := FALSE;
    THIS^.
        AssertEquals_BOOL
    (
        _result
        , sut_readDataNoTag.ReadDataMethod(_udiDataLength, 0).Error
        , 'No Error should be Start Parameter'
    );
END_IF

//Arrange
sut_readDataNoTag();

//Act, Use ReadDataMethod()
sut_readDataNoTag.ReadDataMethod(_udiDataLength, 0);

IF sut_readDataNoTag.isError THEN
    //Assert
    _result := TRUE;

    AssertEquals_BOOL
    (
        _result
        , sut_readDataNoTag.ReadDataMethod(_udiDataLength, 0).Error
        , 'Method did not throw Error'
    );

    AssertEquals_BOOL
    (
        _result
        , sut_readDataNoTag.pReadDataTask.Error
        , 'Task did not throw Error'
    );

    _errorId         := sut_readDataNoTag.ErrorId;
    _expectedErrorId := RFID_FB_U.ERROR.COMMAND_NO_TAG_FOUND;
    AssertEquals(Expected := _expectedErrorId, Actual := _errorId, Message := 'ErrorId must match (No Tag Found)!');

    //Act, Restore(), Error shall disappear
    sut_readDataNoTag.Restore();
    _result := FALSE;

    AssertEquals_BOOL
    (
        _result
        , sut_readDataNoTag.pReadDataTask.Error
        , 'Reset did not Work, Still Status Error'
    );

    _errorId         := sut_readDataNoTag.ErrorId;
    _expectedErrorId := RFID_FB_U.ERROR.NO_ERROR;

    AssertEquals_BOOL
    (
        _result
        , sut_readDataNoTag.pReadDataTask.Error
        , 'Reset did not Work, ErrorID ahs to be No_Error'
    );

    TcUnit.TEST_FINISHED();
END_IF
END_METHOD

METHOD PRIVATE ExecuteReadDataWithOffset_ExpectDataAsString
VAR_INST
    _data          : T_MaxString;
    _expectedData  : T_MaxString := '16# 06 07 08 09'; // Ohne '16# 05 06 07 08' => mit 16# 06 07 08 00
    _result        : BOOL;
    _udiDataLength : uINT := 4;
    _offSet        : BYTE := 1;
END_VAR
//{warning disable C0371}
TcUnit.TEST('ExecuteReadDataWithOffset_ExpectDataAsString');
//Arrange
sut_readDataWithOffset();

//Act

sut_readDataWithOffset.ReadDataMethod(_udiDataLength, _offSet);
//Assert

IF sut_readDataWithOffset.pReadDataTask.Done THEN
    _data := sut_readDataWithOffset.Data;

    AssertEquals_STRING(Expected := _expectedData, Actual := _data, Message := 'Daten passt nicht');

    //Busy off
    _result := FALSE;
    AssertEquals_BOOL
    (
        Expected  := _result
        , Actual  := sut_readDataWithOffset.pReadDataTask.Busy
        , Message := 'Status Busy muss false sein'
    );

    //Status Done mus True sein
    _result := true;
    AssertEquals_BOOL
    (
        Expected  := _result
        , Actual  := sut_readDataWithOffset.ReadDataMethod(_udiDataLength, _offSet).Done
        , Message := 'Status Done muss true sein'
    );

    //Status Done false again
    sut_readDataWithOffset.Restore();
    _result := FALSE;
    AssertEquals_BOOL
    (
        Expected  := _result
        , Actual  := sut_readDataWithOffset.pReadDataTask.Done
        , Message := 'Status Done muss false sein nach Reset'
    );

    TcUnit.TEST_FINISHED();
END_IF
END_METHOD

METHOD PRIVATE ExecuteReadDataWithOffsetTooHigh_ExpectErrorWithErroId
VAR_INST
    _udiDataLength : UINT := 4;
    _offSet        : BYTE := 120;
    _result        : BOOL;
    _firstRun      : BOOL := TRUE;

    _expectedErrorId : RFID_FB_U.ERROR;
    _errorId         : RFID_FB_U.ERROR;

END_VAR
TcUnit.TEST('ExecuteReadDataWithOffsetTooHigh_ExpectErrorWithErroId');
//28 blocks, 4 bytes each, => 112 bytes max user Memory!

//Arrange
sut_readDataWithOffsetTooLong();

//Act, Use ReadDataMethod()
sut_readDataWithOffsetTooLong.ReadDataMethod(udiDataLength := _udiDataLength, MemoryAddr := _offSet);

IF sut_readDataWithOffsetTooLong.pReadDataTask.Error
       OR sut_readUidNoTag.pReadDataTask.Done THEN

    //Assert

    _expectedErrorId := ERROR.COMMAND_ADDRESS_OUTSIDE_TAG_SPECS;
    _errorId         := sut_readDataWithOffsetTooLong.ErrorId;
    AssertEquals(Expected := _expectedErrorId, Actual := _errorId, Message := 'ErrorId must match!');

    _result := TRUE;
    AssertEquals_BOOL
    (
        _result
        , sut_readDataWithOffsetTooLong.ReadDataMethod(_udiDataLength, 0).Error
        , 'Method must throw Error'
    );

    AssertEquals_BOOL
    (
        _result
        , sut_readDataWithOffsetTooLong.pReadDataTask.Error
        , 'Task did not throw Error'
    );

    AssertEquals_BOOL
    (
        _result
        , sut_readDataWithOffsetTooLong.isError
        , 'FB must throw Error'
    );

    //Act, Restore(), Error shall disappear
    sut_readDataWithOffsetTooLong.Restore();
    // more Cycles needed
    sut_readDataWithOffsetTooLong();
    sut_readDataWithOffsetTooLong();
    sut_readDataWithOffsetTooLong();

    _result := FALSE;

    AssertEquals_BOOL
    (
        _result
        , sut_readDataWithOffsetTooLong.IsError
        , 'Reset did not Work, Still Status Error'
    );

    _errorId         := sut_readDataWithOffsetTooLong.ErrorId;
    _expectedErrorId := RFID_FB_U.ERROR.NO_ERROR;
    AssertEquals(Expected := _expectedErrorId, Actual := _errorId, Message := 'ErrorId must match (No Error)!');

    TcUnit.TEST_FINISHED();
END_IF
END_METHOD

METHOD PRIVATE ExecuteReadDataWithTooLongDataLength_ExpectErrorWithErroId
VAR_INST
    _udiDataLength : uINT := 113;
    _result        : BOOL;
    _firstRun      : BOOL := TRUE;

    _expectedErrorId : RFID_FB_U.ERROR;
    _errorId         : RFID_FB_U.ERROR;

END_VAR
TcUnit.TEST('ExecuteReadDataWithTooLongDataLength_ExpectErrorWithErroId');
//28 blocks, 4 bytes each, => 112 bytes max user Memory!

//Arrange
sut_readDataTooLongString();

//Act, Use ReadDataMethod()
sut_readDataTooLongString.ReadDataMethod(udiDataLength := _udiDataLength, MemoryAddr := 0);

IF sut_readDataTooLongString.pReadDataTask.Error
       OR sut_readUidNoTag.pReadDataTask.Done THEN

    //Assert

    _expectedErrorId := ERROR.COMMAND_LENGTH_OUTSIDE_TAG_SPECS;
    _errorId         := sut_readDataTooLongString.ErrorId;
    AssertEquals(Expected := _expectedErrorId, Actual := _errorId, Message := 'ErrorId must match!');

    _result := TRUE;
    AssertEquals_BOOL
    (
        _result
        , sut_readDataTooLongString.ReadDataMethod(_udiDataLength, 0).Error
        , 'Method must throw Error'
    );

    AssertEquals_BOOL
    (
        _result
        , sut_readDataTooLongString.pReadDataTask.Error
        , 'Task did not throw Error'
    );

    AssertEquals_BOOL
    (
        _result
        , sut_readDataTooLongString.isError
        , 'FB must throw Error'
    );

    //Act, Restore(), Error shall disappear
    sut_readDataTooLongString.Restore();
    // more Cycles needed
    sut_readDataTooLongString();
    sut_readDataTooLongString();
    sut_readDataTooLongString();

    _result := FALSE;

    AssertEquals_BOOL
    (
        _result
        , sut_readDataTooLongString.IsError
        , 'Reset did not Work, Still Status Error'
    );

    _errorId         := sut_readDataTooLongString.ErrorId;
    _expectedErrorId := RFID_FB_U.ERROR.NO_ERROR;
    AssertEquals(Expected := _expectedErrorId, Actual := _errorId, Message := 'ErrorId must match (No Error)!');

    TcUnit.TEST_FINISHED();
END_IF
END_METHOD

METHOD ExecuteReadDataWrongParameter_ExpectErrorAndStringError
VAR_INST
    _udiDataLength : UINT := 4;
    _offSet        : BYTE := 120;
    _result        : BOOL;
    _resultString  : STRING := '--Error--';
    _firstRun      : BOOL   := TRUE;

    _expectedErrorId : RFID_FB_U.ERROR;
    _errorId         : RFID_FB_U.ERROR;

END_VAR
TcUnit.TEST('ExecuteReadDataWrongParameter_ExpectErrorAndStringError');

sut_readDataCreateEmptyString();

//Act, Use ReadDataMethod()
sut_readDataCreateEmptyString.ReadDataMethod(udiDataLength := _udiDataLength, MemoryAddr := _offSet);

IF sut_readDataCreateEmptyString.pReadDataTask.Error THEN
    //Assert

    _result := TRUE;
    AssertEquals_BOOL
    (
        _result
        , sut_readDataCreateEmptyString.ReadDataMethod(_udiDataLength, 0).Error
        , 'Method must throw Error'
    );

    AssertEquals_STRING
    (
        Expected  := _resultString
        , actual  := sut_readDataCreateEmptyString.Data
        , Message := 'Data String muss --Error-- sein '
    );

    TcUnit.TEST_FINISHED();
END_IF
END_METHOD

METHOD PRIVATE ExecuteReadUid_ExpectUidAsStringStatusDone
VAR_INST
    _uId         : T_MaxString;
    _expectedUid : T_MaxString := 'E0040150ACF4F3AD';
    _result      : BOOL;
END_VAR
TcUnit.TEST('ExecuteReadUid_ExpectUidAsStringStatusDone');
//Arrange
sut_readUidSuccess();

//Act

sut_readUidSuccess.ReadUidMethod();
//Assert

IF sut_readUidSuccess.pReadUidTask.Done THEN
    _uId := sut_readUidSuccess.Uid;

    AssertEquals_STRING(Expected := _expectedUid, Actual := _uId, Message := 'UID passt nicht');

    //Busy off
    _result := FALSE;
    AssertEquals_BOOL
    (
        Expected  := _result
        , Actual  := sut_readUidSuccess.ReadUidMethod().Busy
        , Message := 'Status Busy muss false sein'
    );

    //Status Done mus True sein
    _result := true;
    AssertEquals_BOOL
    (
        Expected  := _result
        , Actual  := sut_readUidSuccess.ReadUidMethod().Done
        , Message := 'Status Done muss true sein'
    );

    //Status Done false again
    sut_readUidSuccess.Restore();
    _result := FALSE;
    AssertEquals_BOOL
    (
        Expected  := _result
        , Actual  := sut_readUidSuccess.ReadUidMethod().Done
        , Message := 'Status Done muss false sein nach Reset'
    );

    TcUnit.TEST_FINISHED();
END_IF
END_METHOD

METHOD PRIVATE ExecuteReadUidsNoTagInRange_ExpectErrorWithNoTag
VAR_INST
    _udiDataLength : INT := 10;
    _result        : BOOL;
    _firstRun      : BOOL := TRUE;

    _errorId         : RFID_FB_U.ERROR;
    _expectedErrorId : RFID_FB_U.ERROR;

END_VAR
TcUnit.TEST('ExecuteReadUidMethodNoTagInRange_ExpectErrorWithTimeOut');

//Assert Initial State
_result := FALSE;

IF _firstRun THEN
    _firstRun := FALSE;
    THIS^.
        AssertEquals_BOOL
    (
        _result
        , sut_readUidNoTag.ReadUidMethod().Error
        , 'No Error should be Start Parameter'
    );
END_IF

//Arrange
sut_readUidNoTag();

//Act, Use ReadUidMethod()
IF sut_readUidNoTag.ReadUidMethod().Error
       OR sut_readUidNoTag.ReadUidMethod().Done THEN
    //Assert
    _result := TRUE;

    AssertEquals_BOOL
    (
        _result
        , sut_readUidNoTag.ReadUidMethod().Error
        , 'Method did not throw Error'
    );

    AssertEquals_BOOL
    (
        _result
        , sut_readUidNoTag.pReadUidTask.Error
        , 'Task did not throw Error'
    );

    _errorId         := sut_readUidNoTag.ErrorId;
    _expectedErrorId := RFID_FB_U.ERROR.COMMAND_NO_TAG_FOUND;
    AssertEquals(Expected := _expectedErrorId, Actual := _errorId, Message := 'ErrorId must match (No Tag Found)!');

    //Act, Restore(), Error shall disappear
    sut_readUidNoTag.Restore();
    _result := FALSE;

    AssertEquals_BOOL
    (
        _result
        , sut_readUidNoTag.pReadUidTask.Error
        , 'Reset did not Work, Still Status Error'
    );

    TcUnit.TEST_FINISHED();
END_IF
END_METHOD

METHOD PRIVATE ExecuteReadWriteWithOffset_ExpectStatusDone
VAR_INST
    _data          : T_MaxString;
    _expectedData  : T_MaxString := '16# 06 07 08 00'; // Ohne '16# 05 06 07 08' => mit 16# 06 07 08 00
    _result        : BOOL;
    _udiDataLength : uINT := 4;
    _offSet        : BYTE := 1;
END_VAR
//{warning disable C0371}
TcUnit.TEST('ExecuteReadWriteWithOffset_ExpectStatusDone');
//Arrange
sut_writeDataWithOffsetSuccess();

//Act

sut_writeDataWithOffsetSuccess.ReadDataMethod(_udiDataLength, _offSet);
//Assert

IF sut_writeDataWithOffsetSuccess.pReadDataTask.Done THEN
    _data := sut_writeDataWithOffsetSuccess.Data;

    AssertEquals_STRING(Expected := _expectedData, Actual := _data, Message := 'Daten passt nicht');

    //Busy off
    _result := FALSE;
    AssertEquals_BOOL
    (
        Expected  := _result
        , Actual  := sut_writeDataWithOffsetSuccess.pReadDataTask.Busy
        , Message := 'Status Busy muss false sein'
    );

    //Status Done mus True sein
    _result := true;
    AssertEquals_BOOL
    (
        Expected  := _result
        , Actual  := sut_writeDataWithOffsetSuccess.ReadDataMethod(_udiDataLength, _offSet).Done
        , Message := 'Status Done muss true sein'
    );

    //Status Done false again
    sut_writeDataWithOffsetSuccess.Restore();
    _result := FALSE;
    AssertEquals_BOOL
    (
        Expected  := _result
        , Actual  := sut_writeDataWithOffsetSuccess.pReadDataTask.Done
        , Message := 'Status Done muss false sein nach Reset'
    );

    TcUnit.TEST_FINISHED();
END_IF
END_METHOD

METHOD PRIVATE ExecuteWriteData_ExpectStatusDone
VAR_INST
    _testArray : ARRAY[0..4] OF BYTE;

    _result : BOOL;

    _first  : BOOL := TRUE;
    _offSet : BYTE := 1;
END_VAR
TcUnit.TEST('ExecuteWriteData_ExpectStatusDone');
//Arrange
sut_writeDataSuccess();

//Act
sut_writeDataSuccess.WriteDataMethod(WriteData := _testArray, MemoryAddr := 0);

_result := TRUE;

//Needs two Cycles to get from Status Requested to Buisy (TcOpen Framework)
sut_writeDataSuccess();

IF _first THEN
    AssertEquals_BOOL
    (
        Expected  := _result
        , Actual  := sut_writeDataSuccess.pWriteDataTask.Busy
        , Message := 'Status Busy muss true sein'
    );

    _first := FALSE;
END_IF

IF sut_writeDataSuccess.pWriteDataTask.Done THEN

    _result := FALSE;
    AssertEquals_BOOL
    (
        Expected  := _result
        , Actual  := sut_writeDataSuccess.pWriteDataTask.Busy
        , Message := 'Status Busy muss false sein'
    );

    _result := TRUE;
    AssertEquals_BOOL
    (
        Expected  := _result
        , Actual  := sut_writeDataSuccess.WriteDataMethod(WriteData := _testArray, MemoryAddr := 0).Done
        , Message := 'Status Done muss true sein'
    );

    TcUnit.TEST_FINISHED();
END_IF
END_METHOD

PROPERTY Identity : ULINT
GET
Identity := THIS^._nfContext._Identity;
END_GET
END_PROPERTY

PROPERTY Logger : TcoCore.ITcoLogger
GET
Logger := THIS^._nfContext._logger;
END_GET
END_PROPERTY

PROPERTY RealTimeClock : TcoCore.ITcoRtc
GET
RealTimeClock := THIS^._nfContext._rtc;
END_GET
END_PROPERTY

PROPERTY StartCycleCount : ULINT
GET
StartCycleCount := THIS^._nfContext._startCycleCount;
END_GET
END_PROPERTY

END_FUNCTION_BLOCK

// ---- POUs/Turck Rfid Reader/Mock/RfidMockNoRfidInRange.TcPOU
FUNCTION_BLOCK RfidMockNoRfidInRange IMPLEMENTS IRfidHeadWrapper
VAR
    _timeOut        : Tc2_Standard.TON;
    _executionTimer : Tc2_Standard.TON;

    _udintToMillis : UDINT := 1000;
    _busy          : BOOL;

END_VAR

METHOD Execute
VAR_INPUT
    xExecute       : BOOL;
    xAbort         : BOOL;
    udiTimeOut     : UDINT;
    eCommand       : RFID_FB_U.COMMAND;
    udiStartAdress : UDINT;
    uiDataLenght   : UINT;
    myWriteData    : ARRAY[0..127] OF BYTE;
END_VAR
VAR_OUTPUT
    myReadData          : ARRAY[0..127] OF BYTE;
    xDone               : BOOL;
    xBusy               : BOOL;
    xError              : BOOL;
    xAborted            : BOOL;
    eErrorID            : RFID_FB_U.ERROR;
    xTP                 : BOOL;
    xRWHeadNotCOnnected : BOOL;
    uiDataRxLength      : UINT;
END_VAR
IF xExecute THEN
    _busy := TRUE;
END_IF

//28 blocks, 4 bytes each, => 112 bytes max user Memory!
uiDataRxLength := uiDataLenght;
xBusy          := _busy;

_timeOut(in := _busy, PT := UDINT_TO_TIME(udiTimeOut) / _udintToMillis);

xTP := FALSE;

IF _timeOut.Q THEN
    xBusy    := FALSE;
    xError   := TRUE;
    eErrorId := RFID_FB_U.ERROR.TIME_OUT;
END_IF
END_METHOD

END_FUNCTION_BLOCK

// ---- POUs/Turck Rfid Reader/Rfid/RfidHead.TcPOU
FUNCTION_BLOCK RfidHead EXTENDS TcoCore.TcoComponent
VAR_OUTPUT

END_VAR
VAR
    _itfRfidHeadWrapper : IRfidHeadWrapper;
    _readUidTask        : ReadUidTask(THIS^);
    _readDataTask       : ReadDataTask(THIS^);
    _writeDataTask      : WriteDataTask(THIS^);
    _lockTask           : LockTask(THIS^);
    _resetTask          : ResetTaskRfid(THIS^);

    _rfidInOut      : RfidInOut;
    _errorId        : RFID_FB_U.ERROR;
    _uiDataRxLength : UINT;

END_VAR

Map();

_readUidTask(rfidInOut := _rfidInOut, ActionDesc := '<#ReadUid#>');
_readDataTask(rfidInOut := _rfidInOut, ActionDesc := '<#ReadData#>');
_writeDataTask(rfidInOut := _rfidInOut, ActionDesc := '<#WriteData#>');
_lockTask(rfidInOut := _rfidInOut, ActionDesc := '<#WriteData#>');
_resetTask(rfidInOut := _rfidInOut, ActionDesc := '<#ResetTask#>');

PROPERTY Data : Tc2_System.T_MaxString
GET
Data := _readDataTask.Data;
END_GET
END_PROPERTY

PROPERTY DataRxLength : UINT
GET
DataRxLength := _uiDataRxLength;
END_GET
END_PROPERTY

{attribute 'monitoring' := 'call'}
PROPERTY ErrorId : RFID_FB_U.ERROR
GET
{warning disable C0371}
ErrorId := _readDataTask.ErrorId or _readUidTask.ErrorId or _writeDataTask.ErrorId OR _lockTask.ErrorId;
END_GET
END_PROPERTY

METHOD FB_init : BOOL
VAR_INPUT
    bInitRetains       : BOOL; // if TRUE, the retain variables are initialized (warm start / cold start)
    bInCopyCode        : BOOL; // if TRUE, the instance afterwards gets moved into the copy code (online change)
    ParentObject       : ITcoObject;
    itfRfidHeadWrapper : IRfidHeadWrapper;
    udiTimeOut         : TIME;
END_VAR
VAR
    _microToMillis : UDINT := 1000;
END_VAR
// This is not clear to me... I from time to time the consumer code does not see 'FB_init' of 'TcoObject', that's why overridden here with super call...
{warning disable C0316}
SUPER^.FB_init(bInitRetains, bInCopyCode, ParentObject);

THIS^._itfRfidHeadWrapper := itfRfidHeadWrapper;

THIS^._rfidInOut.udiTimeOut := TIME_TO_UDINT(udiTimeOut) * _microToMillis;

_readUidTask.FB_init
(
    bInitRetains   := bInitRetains
    , bInCopyCode  := bInCopyCode
    , ParentObject := ParentObject
);
END_METHOD

{attribute 'monitoring' := 'call'}
PROPERTY IsError : BOOL
GET
//collected Error from Tasks
IsError :=
    this^.pReadUidTask.Error or this^.pReadDataTask.Error or this^.pLockTask.Error or this^.pWriteDataTask.Error;
END_GET
END_PROPERTY

METHOD LockMethod : TcoCore.ITcoTaskStatus
VAR_INPUT
    udiDataLength : UINT;  //Length of the Data to read
    StartAdress   : UDINT; // Memory Adress, from which to start
END_VAR
IF (pLockTask <> 0) THEN
    _rfidInOut.uiDataLenght   := udiDataLength;
    _rfidInOut.udiStartAdress := StartAdress;
    LockMethod                := pLockTask.Invoke();
END_IF
END_METHOD

METHOD Private Map : BOOL
_itfRfidHeadWrapper.Execute
(
    xExecute              := _rfidInOut.xExecute
    , xAbort              := _rfidInOut.xAbort
    , udiTimeOut          := _rfidInOut.udiTimeOut
    , eCommand            := _rfidInOut.eCommand
    , udiStartAdress      := _rfidInOut.udiStartAdress
    , uiDataLenght        := _rfidInOut.uiDataLenght
    , myWriteData         := _rfidInOut.myWriteData
    , myReadData          => _rfidInOut.myReadData
    , xDone               => _rfidInOut.xDone
    , xBusy               => _rfidInOut.xBusy
    , xError              => _rfidInOut.xError
    , xAborted            => _rfidInOut.xAborted
    , eErrorID            => _rfidInOut.eErrorID
    , xTP                 => _rfidInOut.xTP
    , xRWHeadNotCOnnected => _rfidInOut.xRWHeadNotCOnnected
    , uiDataRxLength      => _rfidInOut.uiDataRxLength
);
END_METHOD

PROPERTY pLockTask : TcoCore.ITcoTask
GET
pLockTask := _lockTask;
END_GET
END_PROPERTY

PROPERTY pReadDataTask : TcoCore.ITcoTask
GET
pReadDataTask := _readDataTask;
END_GET
END_PROPERTY

PROPERTY pReadUidTask : TcoCore.ITcoTask
GET
pReadUidTask := _readUidTask;
END_GET
END_PROPERTY

PROPERTY pResetTask : TcoCore.ITcoTask
GET
pResetTask := _resetTask;
END_GET
END_PROPERTY

PROPERTY pWriteDataTask : TcoCore.ITcoTask
GET
pWriteDataTask := _writeDataTask;
END_GET
END_PROPERTY

METHOD ReadDataMethod : TcoCore.ITcoTaskStatus
VAR_INPUT
    udiDataLength : UINT; //Length of the Data to read
    MemoryAddr    : BYTE; // Memory Adress, from which to start
END_VAR
IF (pReadDataTask <> 0) THEN
    _rfidInOut.uiDataLenght   := udiDataLength;
    _rfidInOut.udiStartAdress := MemoryAddr;
    _uiDataRxLength           := _rfidInOut.uiDataRxLength;
    ReadDataMethod            := pReadDataTask.Invoke();
END_IF
END_METHOD

METHOD ReadUidMethod : TcoCore.ITcoTaskStatus
VAR_INPUT
END_VAR
IF (pReadUidTask <> 0) THEN
    ReadUidMethod := pReadUidTask.Invoke();
END_IF
END_METHOD

METHOD ResetMethod : TcoCore.ITcoTaskStatus
IF (pResetTask <> 0) THEN
    ResetMethod := pResetTask.Invoke();
END_IF
END_METHOD

(*~
    <docu>
        <summary>
            Restore all tasks of this instance into initial state.
        </summary>
    </docu>
~*)
METHOD Restore : ITcoRestorable

IF (pReadUidTask <> 0) THEN
    pReadUidTask.Restore();
END_IF;

IF (pReadDataTask <> 0) THEN
    pReadDataTask.Restore();
END_IF;

IF (pWriteDataTask) <> 0 THEN
    pWriteDataTask.Restore();
END_IF

IF (pLockTask) <> 0 THEN
    pLockTask.Restore();
END_IF

IF (pResetTask) <> 0 THEN
    pResetTask.Restore();
END_IF
END_METHOD

METHOD PROTECTED ServiceMode
END_METHOD

PROPERTY Uid : Tc2_System.T_MaxString
GET
Uid := _readUidTask.Uid;
END_GET
END_PROPERTY

METHOD WriteDataMethod : TcoCore.ITcoTaskStatus
VAR_IN_OUT
    WriteData : ARRAY[*] OF BYTE; //Data to write to Tag
END_VAR
VAR_INPUT
    MemoryAddr : BYTE; // Memory Adress, from which to start
END_VAR
VAR_INST
    _i : DINT;
END_VAR
IF (pWriteDataTask <> 0) THEN
    _rfidInOut.uiDataLenght   := SIZEOF(WriteData);
    _rfidInOut.udiStartAdress := MemoryAddr;

    FOR _i := LOWER_BOUND(WriteData, 1) TO UPPER_BOUND(WriteData, 1) DO
        _rfidInOut.myWriteData[_i] := WriteData[_i];
    END_FOR

    _uiDataRxLength := _rfidInOut.uiDataRxLength;
    WriteDataMethod := pWriteDataTask.Invoke();
END_IF
END_METHOD

END_FUNCTION_BLOCK

// ---- POUs/Turck Rfid Reader/Rfid/Tasks/ReadUidTask.TcPOU
FUNCTION_BLOCK ReadUidTask EXTENDS TcoCore.TcoTask
VAR_IN_OUT
    rfidInOut : RfidInOut;
END_VAR
VAR_INPUT
    ActionDesc : STRING(25);
END_VAR

VAR
    _stringBuilder : TcoCore.StringBuilder;
    _state         : INT;
    _coding        : ARRAY[0..7] OF BYTE;
    _index         : INT;
    _hex           : Tc2_System.T_MaxString := '16# ';
    _uidDataLength : UINT                   := 8;

    _eErrorID   : RFID_FB_U.ERROR;
    _noTagFound : BOOL;
    _uid        : Tc2_System.T_MaxString;
END_VAR

IF (THIS^.Execute()) THEN
    THIS^.ThrowWhen(rfidInOut.xError);

    CASE _state OF

        10:
            // Tag vorhanden
            IF NOT rfidInOut.xTP THEN
                THIS^.Messenger.Error
                (
                    _stringBuilder.Append(ActionDesc)
                        .Append('Tag nicht vorhanden bei Leseversuch')
                        .ToString()
                );

                _noTagFound := TRUE;
                ThrowWhen(TRUE);
            ELSE
                _state := 20;
            END_IF
        20:
            //Command setzen
            rfidInOut.eCommand     := command.INVENTORY;
            rfidInOut.uiDataLenght := _uidDataLength;
            _state                 := 30;
        30:
            // Start der Operation
            rfidInOut.xExecute := TRUE;
            _uid               := '';

            _state := 40;
        40:
            // Warte auf Ende Operation
            rfidInOut.myReadData[_index] :=
                (THIS^.rfidInOut.myReadData[_index]);

            IF rfidInOut.xError THEN
                _uid := '--Error--';
            ELSIF rfidInOut.xDone THEN
                FOR _index := 0 TO UINT_TO_INT(rfidInOut.uiDataLenght - 1) DO

                    _uid := Concat
                    (
                        _uid
                        , BYTE_TO_HEXSTR(in := rfidInOut.myReadData[_index], iPrecision := 2, bLoCase := FALSE)
                    );
                END_FOR

                THIS^.DoneWhen(rfidInOut.xDone);
                THIS^.Messenger.Info('Lesen UID erfolgreich');
                _state := 0;
            END_IF
    END_CASE
END_IF

{attribute 'monitoring' := 'call'}
PROPERTY ErrorId : RFID_FB_U.ERROR
GET
{warning disable C0371}
ErrorId := _eErrorID;
END_GET
END_PROPERTY

METHOD PUBLIC FB_init : BOOL
VAR_INPUT
    bInitRetains : BOOL; // if TRUE, the retain variables are initialized (warm start / cold start)
    bInCopyCode  : BOOL; // if TRUE, the instance afterwards gets moved into the copy code (online change)
    ParentObject : ITcoObject;
END_VAR
// This is not clear to me... I from time to time the consumer code does not see 'FB_init' of 'TcoObject', that's why overridden here with super call...
{warning disable C0316}
SUPER^.FB_init(bInitRetains, bInCopyCode, ParentObject);
END_METHOD

(*~
    <docu>
        <summary>
            Executes when task is aborted.
        </summary>
    </docu>
~*)
METHOD PROTECTED OnAbort
{warning disable C0371}
RfidInOut.eCommand := RFID_FB_U.COMMAND.IDLE;
RfidInOut.xExecute := FALSE;
RfidInOut.xAbort   := FALSE;
END_METHOD

(*~
    <docu>
        <summary>
            Executes when task reaches the ```Done``` state .
        </summary>
    </docu>
~*)
METHOD PROTECTED OnDone
{warning disable C0371}
rfidInOut.xExecute := FALSE;
rfidInOut.eCommand := RFID_FB_U.COMMAND.IDLE;
END_METHOD

(*~
    <docu>
        <summary>
            Executes when task reaches the ```Error``` state.
            <para>
                Do not confuse with <see cref="PlcDocu.TcoCore.TcoTask.WhileError()"/>, that is called cyclically until '''Error''' state is left.
            </para>
        </summary>
    </docu>
~*)
METHOD PROTECTED OnError
{warning disable C0371}

IF _noTagFound THEN
    _eErrorID := RFID_FB_U.ERROR.COMMAND_NO_TAG_FOUND;
ELSE
    _eErrorID := rfidInOut.eErrorID;
END_IF

THIS^.Messenger.Build().Append('Rfid Schreib/Lesekopf Fehler : ').Append(to_string(THIS^._eErrorID)).As().AsError();
END_METHOD

(*~
    <docu>
        <summary>
            Executes ones when the task starts (at the moment of transition from the ```Requested``` state into the ```Busy``` state).
        </summary>
    </docu>
~*)
METHOD PROTECTED OnStart
{warning disable C0371}
rfidInOut.eCommand := RFID_FB_U.COMMAND.IDLE;
rfidInOut.xExecute := FALSE;
rfidInOut.xAbort   := FALSE;
_state             := 10;
END_METHOD

(*~
    <docu>
        <summary>
            Restores this instance to the Ready state. Can be called explicitly or from within one of the restore mechanisms.
            <para>
                See also <see cref="PlcDocu.TcoCore.TcoTask.AutoRestorable()"/>
            </para>
        </summary>
    </docu>
~*)
METHOD Restore : ITcoRestorable
{warning disable C0371}
RfidInOut.eCommand := RFID_FB_U.COMMAND.IDLE;
RfidInOut.xExecute := FALSE;
RfidInOut.xAbort   := FALSE;
_eErrorID          := RFID_FB_U.ERROR.NO_ERROR;
SUPER^.Restore();
END_METHOD

PROPERTY Uid : Tc2_System.T_MaxString
GET
Uid := _uId;
END_GET
END_PROPERTY

END_FUNCTION_BLOCK

// ---- POUs/Turck Rfid Reader/Rfid/Tasks/ReadDataTask.TcPOU
FUNCTION_BLOCK ReadDataTask EXTENDS TcoCore.TcoTask
VAR_IN_OUT
    rfidInOut : RfidInOut;
END_VAR
VAR_INPUT
    ActionDesc : STRING(25);
END_VAR
VAR
    _stringBuilder : TcoCore.StringBuilder;
    _state         : INT;
    _coding        : ARRAY[0..3] OF BYTE;
    _index         : INT;
    _hex           : Tc2_System.T_MaxString := '16#';

    _eErrorID   : RFID_FB_U.ERROR;
    _data       : Tc2_System.T_MaxString;
    _noTagFound : BOOL;
END_VAR

IF (THIS^.Execute()) THEN
    THIS^.ThrowWhen(rfidInOut.xError);

    CASE _state OF

        10:
            // Tag vorhanden
            IF NOT rfidInOut.xTP THEN
                THIS^.Messenger.Error
                (
                    _stringBuilder.Append(ActionDesc)
                        .Append('Tag nicht vorhanden bei Leseversuch')
                        .ToString()
                );

                _noTagFound := true;
                ThrowWhen(TRUE);
            ELSE
                _state := 20;
            END_IF
        20:
            //Command setzen
            rfidInOut.eCommand := RFID_FB_U.COMMAND.READ;
            _state             := 30;
        30:
            // Start der Operation
            rfidInOut.xExecute := TRUE;
            _data              := '';

            _state := 40;
        40:
            // Warte auf Ende Operation
            IF rfidInOut.xError THEN
                _data := '--Error--';
            ELSIF rfidInOut.xDone THEN
                FOR _index := 0 TO UINT_TO_INT(rfidInOut.uiDataLenght - 1) DO
                    rfidInOut.myReadData[_index] :=
                        (THIS^.rfidInOut.myReadData[_index]);

                    _data := Concat
                    (
                        _data
                        , Concat
                        (
                            ' '
                            , BYTE_TO_HEXSTR(in := rfidInOut.myReadData[_index], iPrecision := 2, bLoCase := FALSE)
                        )
                    );
                END_FOR

                _data := Concat(_hex, _data);

                THIS^.DoneWhen(rfidInOut.xDone);
                THIS^.Messenger.Info('Lesen der Daten erfolgreich');
                _state := 0;
            END_IF
    END_CASE
END_IF

PROPERTY Data : Tc2_System.T_MaxString
GET
Data := _data;
END_GET
END_PROPERTY

{attribute 'monitoring' := 'call'}
PROPERTY ErrorId : RFID_FB_U.ERROR
GET
{warning disable C0371}
ErrorId := _eErrorID;
END_GET
END_PROPERTY

METHOD PUBLIC FB_init : BOOL
VAR_INPUT
    bInitRetains : BOOL; // if TRUE, the retain variables are initialized (warm start / cold start)
    bInCopyCode  : BOOL; // if TRUE, the instance afterwards gets moved into the copy code (online change)
    ParentObject : ITcoObject;
END_VAR
// This is not clear to me... I from time to time the consumer code does not see 'FB_init' of 'TcoObject', that's why overridden here with super call...
{warning disable C0316}
SUPER^.FB_init(bInitRetains, bInCopyCode, ParentObject);
END_METHOD

(*~
    <docu>
        <summary>
            Executes when task is aborted.
        </summary>
    </docu>
~*)
METHOD PROTECTED OnAbort
{warning disable C0371}
RfidInOut.eCommand := RFID_FB_U.COMMAND.IDLE;
RfidInOut.xExecute := FALSE;
RfidInOut.xAbort   := FALSE;
END_METHOD

(*~
    <docu>
        <summary>
            Executes when task reaches the ```Done``` state .
        </summary>
    </docu>
~*)
METHOD PROTECTED OnDone
{warning disable C0371}
rfidInOut.xExecute := FALSE;
rfidInOut.eCommand := RFID_FB_U.COMMAND.IDLE;
END_METHOD

(*~
    <docu>
        <summary>
            Executes when task reaches the ```Error``` state.
            <para>
                Do not confuse with <see cref="PlcDocu.TcoCore.TcoTask.WhileError()"/>, that is called cyclically until '''Error''' state is left.
            </para>
        </summary>
    </docu>
~*)
METHOD PROTECTED OnError
{warning disable C0371}
IF _noTagFound THEN
    _eErrorID := RFID_FB_U.ERROR.COMMAND_NO_TAG_FOUND;
ELSE
    _eErrorID := rfidInOut.eErrorID;
END_IF

THIS^.Messenger.Build().Append('Rfid Schreib/Lesekopf Fehler : ').Append(to_string(THIS^._eErrorID)).As().AsError();
END_METHOD

(*~
    <docu>
        <summary>
            Executes ones when the task starts (at the moment of transition from the ```Requested``` state into the ```Busy``` state).
        </summary>
    </docu>
~*)
METHOD PROTECTED OnStart
{warning disable C0371}
rfidInOut.eCommand := RFID_FB_U.COMMAND.IDLE;
rfidInOut.xExecute := FALSE;
rfidInOut.xAbort   := FALSE;
_state             := 10;
END_METHOD

(*~
    <docu>
        <summary>
            Restores this instance to the Ready state. Can be called explicitly or from within one of the restore mechanisms.
            <para>
                See also <see cref="PlcDocu.TcoCore.TcoTask.AutoRestorable()"/>
            </para>
        </summary>
    </docu>
~*)
METHOD Restore : ITcoRestorable
{warning disable C0371}
RfidInOut.eCommand := RFID_FB_U.COMMAND.IDLE;
RfidInOut.xExecute := FALSE;
RfidInOut.xAbort   := FALSE;
_noTagFound        := FALSE;
_eErrorID          := RFID_FB_U.ERROR.NO_ERROR;
SUPER^.Restore();
END_METHOD

END_FUNCTION_BLOCK

// ---- POUs/Turck Rfid Reader/Rfid/Tasks/WriteDataTask.TcPOU
FUNCTION_BLOCK WriteDataTask EXTENDS TcoCore.TcoTask
VAR_IN_OUT
    rfidInOut : RfidInOut;
END_VAR
VAR_INPUT
    ActionDesc : STRING(25);
END_VAR
VAR
    _stringBuilder : TcoCore.StringBuilder;
    _state         : INT;

    _eErrorID   : RFID_FB_U.ERROR;
    _data       : Tc2_System.T_MaxString;
    _noTagFound : BOOL;

    _offSet : UDINT;
END_VAR

IF (THIS^.Execute()) THEN
    THIS^.ThrowWhen(rfidInOut.xError);

    CASE _state OF

        10:
            // Tag vorhanden
            IF NOT rfidInOut.xTP THEN
                THIS^.Messenger.Error
                (
                    _stringBuilder.Append(ActionDesc)
                        .Append('Tag nicht vorhanden bei Schreibversuch')
                        .ToString()
                );

                _noTagFound := true;
                ThrowWhen(TRUE);
            ELSE
                _state := 20;
            END_IF
        20:
            //Command setzen
            _offSet            := rfidInOut.udiStartAdress;
            rfidInOut.eCommand := RFID_FB_U.COMMAND.WRITE;
            _state             := 30;
        30:
            // Start der Operation
            rfidInOut.xExecute := TRUE;
            _data              := '';

            _state := 40;
        40:
            // Warte auf Ende Operation
            IF rfidInOut.xError THEN
                ;
            ELSIF rfidInOut.xDone THEN

                THIS^.DoneWhen(rfidInOut.xDone);
                THIS^.Messenger.Info('Schreiben der Daten erfolgreich');
                _state := 0;
            END_IF
    END_CASE
END_IF

{attribute 'monitoring' := 'call'}
PROPERTY ErrorId : RFID_FB_U.ERROR
GET
{warning disable C0371}
ErrorId := _eErrorID;
END_GET
END_PROPERTY

METHOD PUBLIC FB_init : BOOL
VAR_INPUT
    bInitRetains : BOOL; // if TRUE, the retain variables are initialized (warm start / cold start)
    bInCopyCode  : BOOL; // if TRUE, the instance afterwards gets moved into the copy code (online change)
    ParentObject : ITcoObject;
END_VAR
// This is not clear to me... I from time to time the consumer code does not see 'FB_init' of 'TcoObject', that's why overridden here with super call...
{warning disable C0316}
SUPER^.FB_init(bInitRetains, bInCopyCode, ParentObject);
END_METHOD

(*~
    <docu>
        <summary>
            Executes when task is aborted.
        </summary>
    </docu>
~*)
METHOD PROTECTED OnAbort
{warning disable C0371}
RfidInOut.eCommand := RFID_FB_U.COMMAND.IDLE;
RfidInOut.xExecute := FALSE;
RfidInOut.xAbort   := FALSE;
END_METHOD

(*~
    <docu>
        <summary>
            Executes when task reaches the ```Done``` state .
        </summary>
    </docu>
~*)
METHOD PROTECTED OnDone
{warning disable C0371}
rfidInOut.xExecute := FALSE;
rfidInOut.eCommand := RFID_FB_U.COMMAND.IDLE;
END_METHOD

(*~
    <docu>
        <summary>
            Executes when task reaches the ```Error``` state.
            <para>
                Do not confuse with <see cref="PlcDocu.TcoCore.TcoTask.WhileError()"/>, that is called cyclically until '''Error''' state is left.
            </para>
        </summary>
    </docu>
~*)
METHOD PROTECTED OnError
{warning disable C0371}
IF _noTagFound THEN
    _eErrorID := RFID_FB_U.ERROR.COMMAND_NO_TAG_FOUND;
ELSE
    _eErrorID := rfidInOut.eErrorID;
END_IF

THIS^.Messenger.Build().Append('Rfid Schreib/Lesekopf Fehler : ').Append(to_string(THIS^._eErrorID)).As().AsError();
END_METHOD

(*~
    <docu>
        <summary>
            Executes ones when the task starts (at the moment of transition from the ```Requested``` state into the ```Busy``` state).
        </summary>
    </docu>
~*)
METHOD PROTECTED OnStart
{warning disable C0371}
rfidInOut.eCommand := RFID_FB_U.COMMAND.IDLE;
rfidInOut.xExecute := FALSE;
rfidInOut.xAbort   := FALSE;
_state             := 10;
END_METHOD

(*~
    <docu>
        <summary>
            Restores this instance to the Ready state. Can be called explicitly or from within one of the restore mechanisms.
            <para>
                See also <see cref="PlcDocu.TcoCore.TcoTask.AutoRestorable()"/>
            </para>
        </summary>
    </docu>
~*)
METHOD Restore : ITcoRestorable
{warning disable C0371}
RfidInOut.eCommand := RFID_FB_U.COMMAND.IDLE;
RfidInOut.xExecute := FALSE;
RfidInOut.xAbort   := FALSE;
_noTagFound        := FALSE;
_eErrorID          := RFID_FB_U.ERROR.NO_ERROR;
SUPER^.Restore();
END_METHOD

END_FUNCTION_BLOCK

// ---- POUs/Turck Rfid Reader/Rfid/Tasks/LockTask.TcPOU
FUNCTION_BLOCK LockTask EXTENDS TcoCore.TcoTask
VAR_IN_OUT
    rfidInOut : RfidInOut;
END_VAR
VAR_INPUT
    ActionDesc : STRING(25);
END_VAR
VAR
    _stringBuilder : TcoCore.StringBuilder;
    _state         : INT;

    _eErrorID   : RFID_FB_U.ERROR;
    _data       : Tc2_System.T_MaxString;
    _noTagFound : BOOL;

    _offSet : UDINT;
END_VAR

IF (THIS^.Execute()) THEN
    THIS^.ThrowWhen(rfidInOut.xError);

    CASE _state OF

        10:
            // Tag vorhanden
            IF NOT rfidInOut.xTP THEN
                THIS^.Messenger.Error
                (
                    _stringBuilder.Append(ActionDesc)
                        .Append('Tag nicht vorhanden bei Schreibversuch')
                        .ToString()
                );

                _noTagFound := true;
                ThrowWhen(TRUE);
            ELSE
                _state := 20;
            END_IF
        20:
            //Command setzen
            rfidInOut.eCommand := RFID_FB_U.COMMAND.SET_PERMA_LOCK;
            ADSLOGSTR
            (
                msgCtrlMask := ADSLOG_MSGTYPE_ERROR
                , msgFmtStr := 'Startadresse bei CMD: %s'
                , strArg    := TO_STRING(rfidInOut.udiStartAdress)
            );

            _state := 30;
        30:
            // Start der Operation
            rfidInOut.xExecute := TRUE;

            _state := 40;
        40:
            // Warte auf Ende Operation
            IF rfidInOut.xError THEN
                ;
            ELSIF rfidInOut.xDone THEN

                THIS^.DoneWhen(rfidInOut.xDone);
                //                THIS^.Messenger.Info
                //                (
                //                    _stringbuilder.Append('Lock der Daten erfolgreich')
                //                        .Append('Startadresse: ')
                //                        .Append(TO_STRING(rfidinOut.udiStartAdress))
                //                        .Append(' Laenge: ')
                //                        .Append(TO_STRING(rfidInOut.uiDataLenght))
                //                        .ToString()
                //                );
                ADSLOGSTR
                (
                    msgCtrlMask := ADSLOG_MSGTYPE_ERROR
                    , msgFmtStr := 'Startadresse nach Done: %s'
                    , strArg    := TO_STRING(rfidInOut.udiStartAdress)
                );

                _state := 0;
            END_IF
    END_CASE
END_IF

{attribute 'monitoring' := 'call'}
PROPERTY ErrorId : RFID_FB_U.ERROR
GET
{warning disable C0371}
ErrorId := _eErrorID;
END_GET
END_PROPERTY

METHOD PUBLIC FB_init : BOOL
VAR_INPUT
    bInitRetains : BOOL; // if TRUE, the retain variables are initialized (warm start / cold start)
    bInCopyCode  : BOOL; // if TRUE, the instance afterwards gets moved into the copy code (online change)
    ParentObject : ITcoObject;
END_VAR
// This is not clear to me... I from time to time the consumer code does not see 'FB_init' of 'TcoObject', that's why overridden here with super call...
{warning disable C0316}
SUPER^.FB_init(bInitRetains, bInCopyCode, ParentObject);
END_METHOD

(*~
    <docu>
        <summary>
            Executes when task is aborted.
        </summary>
    </docu>
~*)
METHOD PROTECTED OnAbort
{warning disable C0371}
RfidInOut.eCommand := RFID_FB_U.COMMAND.IDLE;
RfidInOut.xExecute := FALSE;
RfidInOut.xAbort   := FALSE;
END_METHOD

(*~
    <docu>
        <summary>
            Executes when task reaches the ```Done``` state .
        </summary>
    </docu>
~*)
METHOD PROTECTED OnDone
{warning disable C0371}
rfidInOut.xExecute := FALSE;
rfidInOut.eCommand := RFID_FB_U.COMMAND.IDLE;
END_METHOD

(*~
    <docu>
        <summary>
            Executes when task reaches the ```Error``` state.
            <para>
                Do not confuse with <see cref="PlcDocu.TcoCore.TcoTask.WhileError()"/>, that is called cyclically until '''Error''' state is left.
            </para>
        </summary>
    </docu>
~*)
METHOD PROTECTED OnError
{warning disable C0371}
IF _noTagFound THEN
    _eErrorID := RFID_FB_U.ERROR.COMMAND_NO_TAG_FOUND;
    // not implemented by Turck
ELSIF rfidInOut.eErrorID = 16#2901 THEN
    _eErrorID := RFID_FB_U.ERROR.COMMAND_ADDRESS_OUTSIDE_BLOCK_BOUNDARIES;
ELSE
    _eErrorID := rfidInOut.eErrorID;
END_IF

THIS^.Messenger.Build().Append('Rfid Schreib/Lesekopf Fehler : ').Append(to_string(THIS^._eErrorID)).As().AsError();
END_METHOD

(*~
    <docu>
        <summary>
            Executes ones when the task starts (at the moment of transition from the ```Requested``` state into the ```Busy``` state).
        </summary>
    </docu>
~*)
METHOD PROTECTED OnStart
{warning disable C0371}
rfidInOut.eCommand := RFID_FB_U.COMMAND.IDLE;
rfidInOut.xExecute := FALSE;
rfidInOut.xAbort   := FALSE;
_state             := 10;
END_METHOD

(*~
    <docu>
        <summary>
            Restores this instance to the Ready state. Can be called explicitly or from within one of the restore mechanisms.
            <para>
                See also <see cref="PlcDocu.TcoCore.TcoTask.AutoRestorable()"/>
            </para>
        </summary>
    </docu>
~*)
METHOD Restore : ITcoRestorable
{warning disable C0371}
RfidInOut.eCommand := RFID_FB_U.COMMAND.IDLE;
RfidInOut.xExecute := FALSE;
RfidInOut.xAbort   := FALSE;
_noTagFound        := FALSE;
_eErrorID          := RFID_FB_U.ERROR.NO_ERROR;
SUPER^.Restore();
END_METHOD

END_FUNCTION_BLOCK

// ---- POUs/Turck Rfid Reader/Rfid/Tasks/ResetTaskRfid.TcPOU
FUNCTION_BLOCK ResetTaskRfid EXTENDS TcoCore.TcoTask
VAR_IN_OUT
    rfidInOut : RfidInOut;
END_VAR
VAR_INPUT
    ActionDesc : STRING(25);
END_VAR
VAR
    _stringBuilder : TcoCore.StringBuilder;
    _state         : INT;

    _eErrorID   : RFID_FB_U.ERROR;
    _data       : Tc2_System.T_MaxString;
    _noTagFound : BOOL;

    _offSet : UDINT;

    _resetResponseCode : UINT := 16#8000;
END_VAR

IF (THIS^.Execute()) THEN

    CASE _state OF

        10:
            _state := 20;

        20:
            //Command setzen
            rfidInOut.eCommand := RFID_FB_U.COMMAND.RESET;
            _state             := 30;
        30:
            // Start der Operation
            rfidInOut.xExecute := TRUE;

